LIN {X 0,Y 346.779,Z 652.941,A -85,B 0,C 180,E1 -23158.009,E2 -23158.009} C_VEL
LIN {X 0,Y 351.853,Z 640.47,A -85,B 0,C 180,E1 -23159.518,E2 -23159.518} C_VEL
LIN {X 0,Y 356.974,Z 626.516,A -85,B 0,C 180,E1 -23160.838,E2 -23160.838} C_VEL
LIN {X 0,Y 360.859,Z 614.191,A -85,B 0,C 180,E1 -23161.77,E2 -23161.77} C_VEL
LIN {X 0,Y 365.059,Z 598.938,A -85,B 0,C 180,E1 -23162.659,E2 -23162.659} C_VEL
LIN {X 0,Y 368.432,Z 583.567,A -85,B 0,C 180,E1 -23163.336,E2 -23163.336} C_VEL
LIN {X 0,Y 383.692,Z 497.433,A -85,B 0,C 180,E1 -23166.383,E2 -23166.383} C_VEL
LIN {X 0,Y 385.575,Z 481.18,A -85,B 0,C 180,E1 -23167.472,E2 -23167.472} C_VEL
LIN {X 0,Y 387.086,Z 465.883,A -85,B 0,C 180,E1 -23168.772,E2 -23168.772} C_VEL
LIN {X 0,Y 387.278,Z 463.542,A -85,B 0,C 180,E1 -23169.013,E2 -23169.013} C_VEL
LIN {X 0,Y 385.216,Z 461.451,A -85,B 0,C 180,E1 -23170.889,E2 -23170.889} C_VEL
LIN {X 0,Y 384.014,Z 460.701,A -85,B 0,C 180,E1 -23172.445,E2 -23172.445} C_VEL
LIN {X 0,Y 383.117,Z 460.948,A -85,B 0,C 180,E1 -23174.518,E2 -23174.518} C_VEL
LIN {X 0,Y 382.898,Z 462.38,A -85,B 0,C 180,E1 -23176.123,E2 -23176.123} C_VEL
LIN {X 0,Y 383.334,Z 465.723,A -85,B 0,C 180,E1 -23178.248,E2 -23178.248} C_VEL
LIN {X 0,Y 384.216,Z 470.909,A -85,B 0,C 180,E1 -23180.158,E2 -23180.158} C_VEL
LIN {X 0,Y 384.484,Z 473.066,A -85,B 0,C 180,E1 -23180.704,E2 -23180.704} C_VEL
LIN {X 0,Y 383.597,Z 487.714,A -85,B 0,C 180,E1 -23182.321,E2 -23182.321} C_VEL
LIN {X 0,Y 382.742,Z 502.862,A -85,B 0,C 180,E1 -23183.728,E2 -23183.728} C_VEL
LIN {X 0,Y 382.412,Z 505.3,A -85,B 0,C 180,E1 -23183.861,E2 -23183.861} C_VEL
LIN {X 0,Y 368.256,Z 585.492,A -85,B 0,C 180,E1 -23186.687,E2 -23186.687} C_VEL
LIN {X 0,Y 365.05,Z 599.465,A -85,B 0,C 180,E1 -23187.34,E2 -23187.34} C_VEL
LIN {X 0,Y 360.944,Z 614.223,A -85,B 0,C 180,E1 -23188.239,E2 -23188.239} C_VEL
LIN {X 0,Y 356.653,Z 627.599,A -85,B 0,C 180,E1 -23189.295,E2 -23189.295} C_VEL
LIN {X 0,Y 352.113,Z 639.917,A -85,B 0,C 180,E1 -23190.506,E2 -23190.506} C_VEL
LIN {X 0,Y 347.039,Z 652.252,A -85,B 0,C 180,E1 -23192.014,E2 -23192.014} C_VEL
LIN {X 0,Y 342.31,Z 662.634,A -85,B 0,C 180,E1 -23193.573,E2 -23193.573} C_VEL
LIN {X 0,Y 337.275,Z 672.679,A -85,B 0,C 180,E1 -23195.459,E2 -23195.459} C_VEL
LIN {X 0,Y 332.699,Z 681,A -85,B 0,C 180,E1 -23197.405,E2 -23197.405} C_VEL
LIN {X 0,Y 328.687,Z 687.815,A -85,B 0,C 180,E1 -23199.414,E2 -23199.414} C_VEL
LIN {X 0,Y 324.702,Z 693.917,A -85,B 0,C 180,E1 -23201.708,E2 -23201.708} C_VEL
LIN {X 0,Y 322.138,Z 697.676,A -85,B 0,C 180,E1 -23203.581,E2 -23203.581} C_VEL
LIN {X 0,Y 319.226,Z 701.269,A -85,B 0,C 180,E1 -23206.033,E2 -23206.033} C_VEL
LIN {X 0,Y 316.907,Z 703.492,A -85,B 0,C 180,E1 -23208.526,E2 -23208.526} C_VEL
LIN {X 0,Y 315.328,Z 704.371,A -85,B 0,C 180,E1 -23211.055,E2 -23211.055} C_VEL
LIN {X 0,Y 314.416,Z 703.91,A -85,B 0,C 180,E1 -23213.605,E2 -23213.605} C_VEL
LIN {X 0,Y 313.985,Z 702.1,A -85,B 0,C 180,E1 -23216.163,E2 -23216.163} C_VEL
LIN {X 0,Y 313.957,Z 698.885,A -85,B 0,C 180,E1 -23218.722,E2 -23218.722} C_VEL
LIN {X 0,Y 314.065,Z 695.439,A -85,B 0,C 180,E1 -23220.639,E2 -23220.639} C_VEL
LIN {X 0,Y 314.17,Z 691.067,A -85,B 0,C 180,E1 -23222.556,E2 -23222.556} C_VEL
LIN {X 0,Y 314.312,Z 684.61,A -85,B 0,C 180,E1 -23224.794,E2 -23224.794} C_VEL
LIN {X 0,Y 314.568,Z 676.533,A -85,B 0,C 180,E1 -23227.035,E2 -23227.035} C_VEL
LIN {X 0,Y 314.911,Z 668.051,A -85,B 0,C 180,E1 -23228.958,E2 -23228.958} C_VEL
LIN {X 0,Y 315.448,Z 657.845,A -85,B 0,C 180,E1 -23230.88,E2 -23230.88} C_VEL
LIN {X 0,Y 316.229,Z 646.555,A -85,B 0,C 180,E1 -23232.635,E2 -23232.635} C_VEL
LIN {X 0,Y 316.961,Z 634.117,A -85,B 0,C 180,E1 -23234.232,E2 -23234.232} C_VEL
LIN {X 0,Y 317.847,Z 620.529,A -85,B 0,C 180,E1 -23235.662,E2 -23235.662} C_VEL
LIN {X 0,Y 318.736,Z 606.233,A -85,B 0,C 180,E1 -23236.847,E2 -23236.847} C_VEL
LIN {X 0,Y 319.44,Z 591.469,A -85,B 0,C 180,E1 -23237.795,E2 -23237.795} C_VEL
LIN {X 0,Y 320.09,Z 576.464,A -85,B 0,C 180,E1 -23238.5,E2 -23238.5} C_VEL
LIN {X 0,Y 323.542,Z 476.916,A -85,B 0,C 180,E1 -23242.075,E2 -23242.075} C_VEL
LIN {X 0,Y 321.24,Z 448.747,A -85,B 0,C 180,E1 -23243.145,E2 -23243.145} C_VEL
LIN {X 0,Y 320.964,Z 439.558,A -85,B 0,C 180,E1 -23243.504,E2 -23243.504} C_VEL
LIN {X 0,Y 323.406,Z 412.958,A -85,B 0,C 180,E1 -23247.629,E2 -23247.629} C_VEL
LIN {X 0,Y 325.023,Z 396.535,A -85,B 0,C 180,E1 -23250.169,E2 -23250.169} C_VEL
LIN {X 0,Y 321.474,Z 379.818,A -85,B 0,C 180,E1 -23253.006,E2 -23253.006} C_VEL
LIN {X 0,Y 316.705,Z 358.595,A -85,B 0,C 180,E1 -23256.736,E2 -23256.736} C_VEL
LIN {X 0,Y 316.607,Z 358.599,A -85,B 0,C 180,E1 -23259.91,E2 -23259.91} C_VEL
LIN {X 0,Y 316.65,Z 358.6,A -85,B 0,C 180,E1 -23263.294,E2 -23263.294} C_VEL
LIN {X 0,Y 316.648,Z 358.598,A -85,B 0,C 180,E1 -23266.885,E2 -23266.885} C_VEL
LIN {X 0,Y 316.625,Z 358.599,A -85,B 0,C 180,E1 -23270.74,E2 -23270.74} C_VEL
LIN {X 0,Y 316.642,Z 358.594,A -85,B 0,C 180,E1 -23273.326,E2 -23273.326} C_VEL
LIN {X 0,Y 316.635,Z 358.596,A -85,B 0,C 180,E1 -23276.424,E2 -23276.424} C_VEL
LIN {X 0,Y 316.649,Z 358.592,A -85,B 0,C 180,E1 -23279.622,E2 -23279.622} C_VEL
LIN {X 0,Y 316.701,Z 358.593,A -85,B 0,C 180,E1 -23283.747,E2 -23283.747} C_VEL
LIN {X 0,Y 316.749,Z 358.588,A -85,B 0,C 180,E1 -23286.371,E2 -23286.371} C_VEL
LIN {X 0,Y 317.718,Z 361.443,A -85,B 0,C 180,E1 -23286.533,E2 -23286.533} C_VEL
LIN {X 0,Y 327.007,Z 380.664,A -85,B 0,C 180,E1 -23287.823,E2 -23287.823} C_VEL
LIN {X 0,Y 332.963,Z 394.934,A -85,B 0,C 180,E1 -23288.65,E2 -23288.65} C_VEL
LIN {X 0,Y 331.321,Z 465.528,A -85,B 0,C 180,E1 -23290.164,E2 -23290.164} C_VEL
LIN {X 0,Y 331.032,Z 481.627,A -85,B 0,C 180,E1 -23290.614,E2 -23290.614} C_VEL
LIN {X 0,Y 330.468,Z 495.129,A -85,B 0,C 180,E1 -23291.222,E2 -23291.222} C_VEL
LIN {X 0,Y 329.533,Z 508.415,A -85,B 0,C 180,E1 -23292.049,E2 -23292.049} C_VEL
LIN {X 0,Y 328.22,Z 521.311,A -85,B 0,C 180,E1 -23293.096,E2 -23293.096} C_VEL
LIN {X 0,Y 326.791,Z 534.282,A -85,B 0,C 180,E1 -23294.459,E2 -23294.459} C_VEL
LIN {X 0,Y 325.343,Z 544.759,A -85,B 0,C 180,E1 -23295.804,E2 -23295.804} C_VEL
LIN {X 0,Y 323.521,Z 555.634,A -85,B 0,C 180,E1 -23297.496,E2 -23297.496} C_VEL
LIN {X 0,Y 321.797,Z 565.3,A -85,B 0,C 180,E1 -23299.338,E2 -23299.338} C_VEL
LIN {X 0,Y 320.333,Z 573.323,A -85,B 0,C 180,E1 -23301.196,E2 -23301.196} C_VEL
LIN {X 0,Y 319.085,Z 580.021,A -85,B 0,C 180,E1 -23303.066,E2 -23303.066} C_VEL
LIN {X 0,Y 318.016,Z 585.608,A -85,B 0,C 180,E1 -23304.946,E2 -23304.946} C_VEL
LIN {X 0,Y 317.008,Z 591.463,A -85,B 0,C 180,E1 -23307.467,E2 -23307.467} C_VEL
LIN {X 0,Y 316.393,Z 595.771,A -85,B 0,C 180,E1 -23310,E2 -23310} C_VEL
LIN {X 0,Y 315.984,Z 598.694,A -85,B 0,C 180,E1 -23312.541,E2 -23312.541} C_VEL
LIN {X 0,Y 316.031,Z 600.28,A -85,B 0,C 180,E1 -23315.086,E2 -23315.086} C_VEL
LIN {X 0,Y 316.305,Z 600.584,A -85,B 0,C 180,E1 -23317.636,E2 -23317.636} C_VEL
LIN {X 0,Y 316.886,Z 599.6,A -85,B 0,C 180,E1 -23320.186,E2 -23320.186} C_VEL
LIN {X 0,Y 317.872,Z 597.292,A -85,B 0,C 180,E1 -23322.73,E2 -23322.73} C_VEL
LIN {X 0,Y 319.35,Z 593.581,A -85,B 0,C 180,E1 -23325.26,E2 -23325.26} C_VEL
LIN {X 0,Y 321.139,Z 588.317,A -85,B 0,C 180,E1 -23327.78,E2 -23327.78} C_VEL
LIN {X 0,Y 322.768,Z 583.279,A -85,B 0,C 180,E1 -23329.656,E2 -23329.656} C_VEL
LIN {X 0,Y 325.037,Z 575.645,A -85,B 0,C 180,E1 -23331.923,E2 -23331.923} C_VEL
LIN {X 0,Y 327.491,Z 566.918,A -85,B 0,C 180,E1 -23333.978,E2 -23333.978} C_VEL
LIN {X 0,Y 329.941,Z 557.378,A -85,B 0,C 180,E1 -23335.799,E2 -23335.799} C_VEL
LIN {X 0,Y 332.282,Z 546.761,A -85,B 0,C 180,E1 -23337.46,E2 -23337.46} C_VEL
LIN {X 0,Y 334.603,Z 534.957,A -85,B 0,C 180,E1 -23338.953,E2 -23338.953} C_VEL
LIN {X 0,Y 336.61,Z 523.311,A -85,B 0,C 180,E1 -23340.134,E2 -23340.134} C_VEL
LIN {X 0,Y 338.141,Z 510.547,A -85,B 0,C 180,E1 -23341.189,E2 -23341.189} C_VEL
LIN {X 0,Y 339.438,Z 497.149,A -85,B 0,C 180,E1 -23342.03,E2 -23342.03} C_VEL
LIN {X 0,Y 340.324,Z 482.787,A -85,B 0,C 180,E1 -23342.674,E2 -23342.674} C_VEL
LIN {X 0,Y 340.732,Z 467.217,A -85,B 0,C 180,E1 -23343.114,E2 -23343.114} C_VEL
LIN {X 0,Y 342.688,Z 407.141,A -85,B 0,C 180,E1 -23344.365,E2 -23344.365} C_VEL
LIN {X 0,Y 334.807,Z 391.079,A -85,B 0,C 180,E1 -23345.625,E2 -23345.625} C_VEL
LIN {X 0,Y 324.967,Z 373.249,A -85,B 0,C 180,E1 -23347.256,E2 -23347.256} C_VEL
LIN {X 0,Y 318.296,Z 362.362,A -85,B 0,C 180,E1 -23348.406,E2 -23348.406} C_VEL
LIN {X 0,Y 316.879,Z 359.863,A -85,B 0,C 180,E1 -23348.664,E2 -23348.664} C_VEL
LIN {X 0,Y 316.605,Z 358.608,A -85,B 0,C 180,E1 -23348.766,E2 -23348.766} C_VEL
LIN {X 0,Y 316.591,Z 358.608,A -85,B 0,C 180,E1 -23351.586,E2 -23351.586} C_VEL
LIN {X 0,Y 316.61,Z 358.6,A -85,B 0,C 180,E1 -23355.068,E2 -23355.068} C_VEL
LIN {X 0,Y 316.606,Z 358.602,A -85,B 0,C 180,E1 -23358.782,E2 -23358.782} C_VEL
LIN {X 0,Y 316.63,Z 358.554,A -85,B 0,C 180,E1 -23362.787,E2 -23362.787} C_VEL
LIN {X 0,Y 316.621,Z 358.596,A -85,B 0,C 180,E1 -23366.422,E2 -23366.422} C_VEL
LIN {X 0,Y 316.626,Z 358.587,A -85,B 0,C 180,E1 -23369.629,E2 -23369.629} C_VEL
LIN {X 0,Y 316.684,Z 358.581,A -85,B 0,C 180,E1 -23373.745,E2 -23373.745} C_VEL
LIN {X 0,Y 316.719,Z 358.59,A -85,B 0,C 180,E1 -23376.824,E2 -23376.824} C_VEL
LIN {X 0,Y 322.641,Z 381.681,A -85,B 0,C 180,E1 -23377.798,E2 -23377.798} C_VEL
LIN {X 0,Y 322.664,Z 387.019,A -85,B 0,C 180,E1 -23377.988,E2 -23377.988} C_VEL
LIN {X 0,Y 321.766,Z 392.772,A -85,B 0,C 180,E1 -23378.173,E2 -23378.173} C_VEL
LIN {X 0,Y 315.268,Z 411.293,A -85,B 0,C 180,E1 -23378.723,E2 -23378.723} C_VEL
LIN {X 0,Y 314.476,Z 417.043,A -85,B 0,C 180,E1 -23378.922,E2 -23378.922} C_VEL
LIN {X 0,Y 313.091,Z 476.776,A -85,B 0,C 180,E1 -23381.113,E2 -23381.113} C_VEL
LIN {X 0,Y 312.579,Z 491.416,A -85,B 0,C 180,E1 -23381.885,E2 -23381.885} C_VEL
LIN {X 0,Y 312.014,Z 505.448,A -85,B 0,C 180,E1 -23382.863,E2 -23382.863} C_VEL
LIN {X 0,Y 311.237,Z 520.037,A -85,B 0,C 180,E1 -23384.164,E2 -23384.164} C_VEL
LIN {X 0,Y 310.556,Z 533.361,A -85,B 0,C 180,E1 -23385.635,E2 -23385.635} C_VEL
LIN {X 0,Y 309.939,Z 545.605,A -85,B 0,C 180,E1 -23387.27,E2 -23387.27} C_VEL
LIN {X 0,Y 309.213,Z 557.66,A -85,B 0,C 180,E1 -23389.229,E2 -23389.229} C_VEL
LIN {X 0,Y 308.697,Z 567.679,A -85,B 0,C 180,E1 -23391.19,E2 -23391.19} C_VEL
LIN {X 0,Y 308.33,Z 577.376,A -85,B 0,C 180,E1 -23393.478,E2 -23393.478} C_VEL
LIN {X 0,Y 308.286,Z 585.271,A -85,B 0,C 180,E1 -23395.765,E2 -23395.765} C_VEL
LIN {X 0,Y 308.365,Z 591.806,A -85,B 0,C 180,E1 -23398.112,E2 -23398.112} C_VEL
LIN {X 0,Y 308.83,Z 597.364,A -85,B 0,C 180,E1 -23400.649,E2 -23400.649} C_VEL
LIN {X 0,Y 309.447,Z 600.59,A -85,B 0,C 180,E1 -23402.594,E2 -23402.594} C_VEL
LIN {X 0,Y 310.787,Z 603.654,A -85,B 0,C 180,E1 -23405.172,E2 -23405.172} C_VEL
LIN {X 0,Y 312.509,Z 605.336,A -85,B 0,C 180,E1 -23407.728,E2 -23407.728} C_VEL
LIN {X 0,Y 314.673,Z 605.643,A -85,B 0,C 180,E1 -23410.257,E2 -23410.257} C_VEL
LIN {X 0,Y 317.708,Z 604.49,A -85,B 0,C 180,E1 -23412.736,E2 -23412.736} C_VEL
LIN {X 0,Y 321.376,Z 601.907,A -85,B 0,C 180,E1 -23415.161,E2 -23415.161} C_VEL
LIN {X 0,Y 325.315,Z 597.923,A -85,B 0,C 180,E1 -23417.544,E2 -23417.544} C_VEL
LIN {X 0,Y 328.569,Z 593.917,A -85,B 0,C 180,E1 -23419.295,E2 -23419.295} C_VEL
LIN {X 0,Y 333.406,Z 587.105,A -85,B 0,C 180,E1 -23421.571,E2 -23421.571} C_VEL
LIN {X 0,Y 337.979,Z 579.557,A -85,B 0,C 180,E1 -23423.512,E2 -23423.512} C_VEL
LIN {X 0,Y 342.881,Z 570.267,A -85,B 0,C 180,E1 -23425.403,E2 -23425.403} C_VEL
LIN {X 0,Y 347.411,Z 560.641,A -85,B 0,C 180,E1 -23426.977,E2 -23426.977} C_VEL
LIN {X 0,Y 352.14,Z 549.032,A -85,B 0,C 180,E1 -23428.515,E2 -23428.515} C_VEL
LIN {X 0,Y 356.656,Z 536.172,A -85,B 0,C 180,E1 -23429.89,E2 -23429.89} C_VEL
LIN {X 0,Y 360.336,Z 523.4,A -85,B 0,C 180,E1 -23431.006,E2 -23431.006} C_VEL
LIN {X 0,Y 363.682,Z 509.402,A -85,B 0,C 180,E1 -23431.981,E2 -23431.981} C_VEL
LIN {X 0,Y 366.369,Z 495.047,A -85,B 0,C 180,E1 -23432.767,E2 -23432.767} C_VEL
LIN {X 0,Y 370.41,Z 469.275,A -85,B 0,C 180,E1 -23433.806,E2 -23433.806} C_VEL
LIN {X 0,Y 375.351,Z 441.241,A -85,B 0,C 180,E1 -23434.806,E2 -23434.806} C_VEL
LIN {X 0,Y 373.14,Z 436.29,A -85,B 0,C 180,E1 -23436.453,E2 -23436.453} C_VEL
LIN {X 0,Y 371.66,Z 433.21,A -85,B 0,C 180,E1 -23437.804,E2 -23437.804} C_VEL
LIN {X 0,Y 370.173,Z 429.982,A -85,B 0,C 180,E1 -23439.676,E2 -23439.676} C_VEL
LIN {X 0,Y 368.834,Z 428.602,A -85,B 0,C 180,E1 -23442.214,E2 -23442.214} C_VEL
LIN {X 0,Y 368.77,Z 428.453,A -85,B 0,C 180,E1 -23444.198,E2 -23444.198} C_VEL
LIN {X 0,Y 369.948,Z 429.972,A -85,B 0,C 180,E1 -23447.03,E2 -23447.03} C_VEL
LIN {X 0,Y 371.094,Z 432.974,A -85,B 0,C 180,E1 -23448.705,E2 -23448.705} C_VEL
LIN {X 0,Y 371.308,Z 443.447,A -85,B 0,C 180,E1 -23450.524,E2 -23450.524} C_VEL
LIN {X 0,Y 370.005,Z 459.779,A -85,B 0,C 180,E1 -23451.954,E2 -23451.954} C_VEL
LIN {X 0,Y 368.744,Z 476.184,A -85,B 0,C 180,E1 -23453.226,E2 -23453.226} C_VEL
LIN {X 0,Y 367.73,Z 487.498,A -85,B 0,C 180,E1 -23453.981,E2 -23453.981} C_VEL
LIN {X 0,Y 366.638,Z 496.863,A -85,B 0,C 180,E1 -23454.488,E2 -23454.488} C_VEL
LIN {X 0,Y 360.902,Z 530.902,A -85,B 0,C 180,E1 -23455.705,E2 -23455.705} C_VEL
LIN {X 0,Y 356.785,Z 548.297,A -85,B 0,C 180,E1 -23456.485,E2 -23456.485} C_VEL
LIN {X 0,Y 352.248,Z 563.594,A -85,B 0,C 180,E1 -23457.358,E2 -23457.358} C_VEL
LIN {X 0,Y 347.42,Z 577.531,A -85,B 0,C 180,E1 -23458.386,E2 -23458.386} C_VEL
LIN {X 0,Y 341.838,Z 591.573,A -85,B 0,C 180,E1 -23459.696,E2 -23459.696} C_VEL
LIN {X 0,Y 336.493,Z 603.77,A -85,B 0,C 180,E1 -23461.124,E2 -23461.124} C_VEL
LIN {X 0,Y 331.55,Z 614.197,A -85,B 0,C 180,E1 -23462.645,E2 -23462.645} C_VEL
LIN {X 0,Y 326.244,Z 624.904,A -85,B 0,C 180,E1 -23464.57,E2 -23464.57} C_VEL
LIN {X 0,Y 321.587,Z 633.763,A -85,B 0,C 180,E1 -23466.578,E2 -23466.578} C_VEL
LIN {X 0,Y 317.657,Z 641.179,A -85,B 0,C 180,E1 -23468.664,E2 -23468.664} C_VEL
LIN {X 0,Y 314.652,Z 646.488,A -85,B 0,C 180,E1 -23470.493,E2 -23470.493} C_VEL
LIN {X 0,Y 311.633,Z 652.249,A -85,B 0,C 180,E1 -23473.01,E2 -23473.01} C_VEL
LIN {X 0,Y 309.58,Z 656.596,A -85,B 0,C 180,E1 -23475.588,E2 -23475.588} C_VEL
LIN {X 0,Y 308.34,Z 659.625,A -85,B 0,C 180,E1 -23478.202,E2 -23478.202} C_VEL
LIN {X 0,Y 308.143,Z 660.826,A -85,B 0,C 180,E1 -23479.729,E2 -23479.729} C_VEL
LIN {X 0,Y 307.758,Z 669.853,A -85,B 0,C 180,E1 -23481.492,E2 -23481.492} C_VEL
LIN {X 0,Y 307.479,Z 678.288,A -85,B 0,C 180,E1 -23483.46,E2 -23483.46} C_VEL
LIN {X 0,Y 307.33,Z 686.328,A -85,B 0,C 180,E1 -23485.752,E2 -23485.752} C_VEL
LIN {X 0,Y 307.193,Z 692.677,A -85,B 0,C 180,E1 -23488.04,E2 -23488.04} C_VEL
LIN {X 0,Y 307.15,Z 696.963,A -85,B 0,C 180,E1 -23490,E2 -23490} C_VEL
LIN {X 0,Y 306.964,Z 701.209,A -85,B 0,C 180,E1 -23492.616,E2 -23492.616} C_VEL
LIN {X 0,Y 307.071,Z 703.981,A -85,B 0,C 180,E1 -23495.235,E2 -23495.235} C_VEL
LIN {X 0,Y 307.682,Z 705.368,A -85,B 0,C 180,E1 -23497.85,E2 -23497.85} C_VEL
LIN {X 0,Y 308.888,Z 705.414,A -85,B 0,C 180,E1 -23500.452,E2 -23500.452} C_VEL
LIN {X 0,Y 310.84,Z 704.125,A -85,B 0,C 180,E1 -23503.023,E2 -23503.023} C_VEL
LIN {X 0,Y 313.636,Z 701.476,A -85,B 0,C 180,E1 -23505.545,E2 -23505.545} C_VEL
LIN {X 0,Y 316.707,Z 697.478,A -85,B 0,C 180,E1 -23508.037,E2 -23508.037} C_VEL
LIN {X 0,Y 320.721,Z 691.969,A -85,B 0,C 180,E1 -23510.453,E2 -23510.453} C_VEL
LIN {X 0,Y 325.464,Z 684.838,A -85,B 0,C 180,E1 -23512.792,E2 -23512.792} C_VEL
LIN {X 0,Y 330.082,Z 677.116,A -85,B 0,C 180,E1 -23514.778,E2 -23514.778} C_VEL
LIN {X 0,Y 335.287,Z 667.758,A -85,B 0,C 180,E1 -23516.689,E2 -23516.689} C_VEL
LIN {X 0,Y 340.088,Z 658.186,A -85,B 0,C 180,E1 -23518.275,E2 -23518.275} C_VEL
LIN {X 0,Y 345.725,Z 645.746,A -85,B 0,C 180,E1 -23519.928,E2 -23519.928} C_VEL
LIN {X 0,Y 350.346,Z 634.318,A -85,B 0,C 180,E1 -23521.152,E2 -23521.152} C_VEL
LIN {X 0,Y 355.301,Z 620.631,A -85,B 0,C 180,E1 -23522.327,E2 -23522.327} C_VEL
LIN {X 0,Y 360.184,Z 604.828,A -85,B 0,C 180,E1 -23523.357,E2 -23523.357} C_VEL
LIN {X 0,Y 363.719,Z 591.16,A -85,B 0,C 180,E1 -23524.034,E2 -23524.034} C_VEL
LIN {X 0,Y 367.59,Z 571.441,A -85,B 0,C 180,E1 -23524.782,E2 -23524.782} C_VEL
LIN {X 0,Y 381.113,Z 498.793,A -85,B 0,C 180,E1 -23527.362,E2 -23527.362} C_VEL
LIN {X 0,Y 383.099,Z 483.725,A -85,B 0,C 180,E1 -23528.391,E2 -23528.391} C_VEL
LIN {X 0,Y 384.77,Z 469.789,A -85,B 0,C 180,E1 -23529.579,E2 -23529.579} C_VEL
LIN {X 0,Y 383.357,Z 468.269,A -85,B 0,C 180,E1 -23530.972,E2 -23530.972} C_VEL
LIN {X 0,Y 382.078,Z 467.548,A -85,B 0,C 180,E1 -23532.711,E2 -23532.711} C_VEL
LIN {X 0,Y 381.318,Z 467.919,A -85,B 0,C 180,E1 -23534.616,E2 -23534.616} C_VEL
LIN {X 0,Y 381.122,Z 469.709,A -85,B 0,C 180,E1 -23536.392,E2 -23536.392} C_VEL
LIN {X 0,Y 381.417,Z 472.559,A -85,B 0,C 180,E1 -23538.079,E2 -23538.079} C_VEL
LIN {X 0,Y 382.066,Z 477.105,A -85,B 0,C 180,E1 -23539.76,E2 -23539.76} C_VEL
LIN {X 0,Y 382.12,Z 478.457,A -85,B 0,C 180,E1 -23540.064,E2 -23540.064} C_VEL
LIN {X 0,Y 380.815,Z 494.198,A -85,B 0,C 180,E1 -23541.784,E2 -23541.784} C_VEL
LIN {X 0,Y 379.927,Z 505.742,A -85,B 0,C 180,E1 -23542.854,E2 -23542.854} C_VEL
LIN {X 0,Y 367.019,Z 575.904,A -85,B 0,C 180,E1 -23545.322,E2 -23545.322} C_VEL
LIN {X 0,Y 363.346,Z 593.162,A -85,B 0,C 180,E1 -23546.01,E2 -23546.01} C_VEL
LIN {X 0,Y 359.038,Z 609.143,A -85,B 0,C 180,E1 -23546.89,E2 -23546.89} C_VEL
LIN {X 0,Y 354.944,Z 621.931,A -85,B 0,C 180,E1 -23547.804,E2 -23547.804} C_VEL
LIN {X 0,Y 350.056,Z 635.127,A -85,B 0,C 180,E1 -23548.986,E2 -23548.986} C_VEL
LIN {X 0,Y 345.053,Z 647.242,A -85,B 0,C 180,E1 -23550.343,E2 -23550.343} C_VEL
LIN {X 0,Y 340.342,Z 657.483,A -85,B 0,C 180,E1 -23551.748,E2 -23551.748} C_VEL
LIN {X 0,Y 334.758,Z 668.398,A -85,B 0,C 180,E1 -23553.6,E2 -23553.6} C_VEL
LIN {X 0,Y 329.702,Z 677.411,A -85,B 0,C 180,E1 -23555.527,E2 -23555.527} C_VEL
LIN {X 0,Y 325.727,Z 683.918,A -85,B 0,C 180,E1 -23557.228,E2 -23557.228} C_VEL
LIN {X 0,Y 321.099,Z 690.959,A -85,B 0,C 180,E1 -23559.573,E2 -23559.573} C_VEL
LIN {X 0,Y 316.996,Z 696.44,A -85,B 0,C 180,E1 -23561.98,E2 -23561.98} C_VEL
LIN {X 0,Y 313.898,Z 700.4,A -85,B 0,C 180,E1 -23564.469,E2 -23564.469} C_VEL
LIN {X 0,Y 311.068,Z 703.028,A -85,B 0,C 180,E1 -23566.987,E2 -23566.987} C_VEL
LIN {X 0,Y 309.051,Z 704.298,A -85,B 0,C 180,E1 -23569.554,E2 -23569.554} C_VEL
LIN {X 0,Y 307.759,Z 704.237,A -85,B 0,C 180,E1 -23572.152,E2 -23572.152} C_VEL
LIN {X 0,Y 307.078,Z 702.839,A -85,B 0,C 180,E1 -23574.765,E2 -23574.765} C_VEL
LIN {X 0,Y 306.869,Z 700.065,A -85,B 0,C 180,E1 -23577.384,E2 -23577.384} C_VEL
LIN {X 0,Y 306.986,Z 695.832,A -85,B 0,C 180,E1 -23580,E2 -23580} C_VEL
LIN {X 0,Y 307.097,Z 691.59,A -85,B 0,C 180,E1 -23581.961,E2 -23581.961} C_VEL
LIN {X 0,Y 307.279,Z 685.311,A -85,B 0,C 180,E1 -23584.249,E2 -23584.249} C_VEL
LIN {X 0,Y 307.46,Z 677.251,A -85,B 0,C 180,E1 -23586.576,E2 -23586.576} C_VEL
LIN {X 0,Y 307.848,Z 667.58,A -85,B 0,C 180,E1 -23588.835,E2 -23588.835} C_VEL
LIN {X 0,Y 308.407,Z 657.294,A -85,B 0,C 180,E1 -23590.8,E2 -23590.8} C_VEL
LIN {X 0,Y 309.188,Z 645.655,A -85,B 0,C 180,E1 -23592.635,E2 -23592.635} C_VEL
LIN {X 0,Y 309.896,Z 633.374,A -85,B 0,C 180,E1 -23594.23,E2 -23594.23} C_VEL
LIN {X 0,Y 310.831,Z 619.593,A -85,B 0,C 180,E1 -23595.689,E2 -23595.689} C_VEL
LIN {X 0,Y 311.678,Z 605.115,A -85,B 0,C 180,E1 -23596.903,E2 -23596.903} C_VEL
LIN {X 0,Y 312.371,Z 590.156,A -85,B 0,C 180,E1 -23597.874,E2 -23597.874} C_VEL
LIN {X 0,Y 313.093,Z 573.682,A -85,B 0,C 180,E1 -23598.633,E2 -23598.633} C_VEL
LIN {X 0,Y 316.466,Z 477.377,A -85,B 0,C 180,E1 -23602.199,E2 -23602.199} C_VEL
LIN {X 0,Y 314.199,Z 448.926,A -85,B 0,C 180,E1 -23603.31,E2 -23603.31} C_VEL
LIN {X 0,Y 313.934,Z 439.598,A -85,B 0,C 180,E1 -23603.68,E2 -23603.68} C_VEL
LIN {X 0,Y 316.358,Z 414.017,A -85,B 0,C 180,E1 -23607.708,E2 -23607.708} C_VEL
LIN {X 0,Y 317.988,Z 397.796,A -85,B 0,C 180,E1 -23610.257,E2 -23610.257} C_VEL
LIN {X 0,Y 315.094,Z 383.863,A -85,B 0,C 180,E1 -23612.654,E2 -23612.654} C_VEL
LIN {X 0,Y 310.71,Z 364.228,A -85,B 0,C 180,E1 -23616.117,E2 -23616.117} C_VEL
LIN {X 0,Y 309.662,Z 359.473,A -85,B 0,C 180,E1 -23616.997,E2 -23616.997} C_VEL
LIN {X 0,Y 309.591,Z 359.473,A -85,B 0,C 180,E1 -23621.005,E2 -23621.005} C_VEL
LIN {X 0,Y 309.61,Z 359.476,A -85,B 0,C 180,E1 -23624.534,E2 -23624.534} C_VEL
LIN {X 0,Y 309.593,Z 359.478,A -85,B 0,C 180,E1 -23628.299,E2 -23628.299} C_VEL
LIN {X 0,Y 309.609,Z 359.477,A -85,B 0,C 180,E1 -23632.357,E2 -23632.357} C_VEL
LIN {X 0,Y 309.593,Z 359.476,A -85,B 0,C 180,E1 -23635.555,E2 -23635.555} C_VEL
LIN {X 0,Y 309.606,Z 359.464,A -85,B 0,C 180,E1 -23639.284,E2 -23639.284} C_VEL
LIN {X 0,Y 309.641,Z 359.473,A -85,B 0,C 180,E1 -23643.101,E2 -23643.101} C_VEL
LIN {X 0,Y 309.669,Z 359.469,A -85,B 0,C 180,E1 -23645.699,E2 -23645.699} C_VEL
LIN {X 0,Y 310.783,Z 362.472,A -85,B 0,C 180,E1 -23645.904,E2 -23645.904} C_VEL
LIN {X 0,Y 320.548,Z 382.539,A -85,B 0,C 180,E1 -23647.309,E2 -23647.309} C_VEL
LIN {X 0,Y 326.56,Z 396.904,A -85,B 0,C 180,E1 -23648.173,E2 -23648.173} C_VEL
LIN {X 0,Y 324.818,Z 464.966,A -85,B 0,C 180,E1 -23649.652,E2 -23649.652} C_VEL
LIN {X 0,Y 324.54,Z 480.842,A -85,B 0,C 180,E1 -23650.087,E2 -23650.087} C_VEL
LIN {X 0,Y 323.967,Z 494.854,A -85,B 0,C 180,E1 -23650.707,E2 -23650.707} C_VEL
LIN {X 0,Y 322.977,Z 508.959,A -85,B 0,C 180,E1 -23651.59,E2 -23651.59} C_VEL
LIN {X 0,Y 321.687,Z 521.072,A -85,B 0,C 180,E1 -23652.579,E2 -23652.579} C_VEL
LIN {X 0,Y 320.379,Z 532.973,A -85,B 0,C 180,E1 -23653.814,E2 -23653.814} C_VEL
LIN {X 0,Y 318.861,Z 543.972,A -85,B 0,C 180,E1 -23655.21,E2 -23655.21} C_VEL
LIN {X 0,Y 316.995,Z 554.996,A -85,B 0,C 180,E1 -23656.91,E2 -23656.91} C_VEL
LIN {X 0,Y 315.153,Z 564.901,A -85,B 0,C 180,E1 -23658.786,E2 -23658.786} C_VEL
LIN {X 0,Y 313.611,Z 573.123,A -85,B 0,C 180,E1 -23660.681,E2 -23660.681} C_VEL
LIN {X 0,Y 312.091,Z 580.985,A -85,B 0,C 180,E1 -23662.91,E2 -23662.91} C_VEL
LIN {X 0,Y 311.005,Z 586.539,A -85,B 0,C 180,E1 -23664.832,E2 -23664.832} C_VEL
LIN {X 0,Y 309.978,Z 592.35,A -85,B 0,C 180,E1 -23667.41,E2 -23667.41} C_VEL
LIN {X 0,Y 309.325,Z 596.627,A -85,B 0,C 180,E1 -23670,E2 -23670} C_VEL
LIN {X 0,Y 308.935,Z 599.516,A -85,B 0,C 180,E1 -23672.599,E2 -23672.599} C_VEL
LIN {X 0,Y 308.995,Z 601.071,A -85,B 0,C 180,E1 -23675.203,E2 -23675.203} C_VEL
LIN {X 0,Y 309.288,Z 601.346,A -85,B 0,C 180,E1 -23677.81,E2 -23677.81} C_VEL
LIN {X 0,Y 309.908,Z 600.331,A -85,B 0,C 180,E1 -23680.417,E2 -23680.417} C_VEL
LIN {X 0,Y 310.971,Z 597.989,A -85,B 0,C 180,E1 -23683.017,E2 -23683.017} C_VEL
LIN {X 0,Y 312.483,Z 594.241,A -85,B 0,C 180,E1 -23685.604,E2 -23685.604} C_VEL
LIN {X 0,Y 314.358,Z 588.93,A -85,B 0,C 180,E1 -23688.177,E2 -23688.177} C_VEL
LIN {X 0,Y 316.061,Z 583.869,A -85,B 0,C 180,E1 -23690.091,E2 -23690.091} C_VEL
LIN {X 0,Y 318.33,Z 576.573,A -85,B 0,C 180,E1 -23692.298,E2 -23692.298} C_VEL
LIN {X 0,Y 320.604,Z 568.858,A -85,B 0,C 180,E1 -23694.183,E2 -23694.183} C_VEL
LIN {X 0,Y 323.088,Z 559.56,A -85,B 0,C 180,E1 -23696.041,E2 -23696.041} C_VEL
LIN {X 0,Y 325.558,Z 549.225,A -85,B 0,C 180,E1 -23697.728,E2 -23697.728} C_VEL
LIN {X 0,Y 327.647,Z 539.067,A -85,B 0,C 180,E1 -23699.101,E2 -23699.101} C_VEL
LIN {X 0,Y 329.966,Z 526.602,A -85,B 0,C 180,E1 -23700.452,E2 -23700.452} C_VEL
LIN {X 0,Y 331.604,Z 514.494,A -85,B 0,C 180,E1 -23701.52,E2 -23701.52} C_VEL
LIN {X 0,Y 333.051,Z 500.538,A -85,B 0,C 180,E1 -23702.47,E2 -23702.47} C_VEL
LIN {X 0,Y 334.067,Z 486.744,A -85,B 0,C 180,E1 -23703.148,E2 -23703.148} C_VEL
LIN {X 0,Y 334.552,Z 472.312,A -85,B 0,C 180,E1 -23703.623,E2 -23703.623} C_VEL
LIN {X 0,Y 336.632,Z 409.302,A -85,B 0,C 180,E1 -23704.965,E2 -23704.965} C_VEL
LIN {X 0,Y 329.186,Z 394.16,A -85,B 0,C 180,E1 -23706.198,E2 -23706.198} C_VEL
LIN {X 0,Y 319.879,Z 377.285,A -85,B 0,C 180,E1 -23707.792,E2 -23707.792} C_VEL
LIN {X 0,Y 311.554,Z 363.621,A -85,B 0,C 180,E1 -23709.288,E2 -23709.288} C_VEL
LIN {X 0,Y 309.943,Z 361.107,A -85,B 0,C 180,E1 -23709.587,E2 -23709.587} C_VEL
LIN {X 0,Y 309.523,Z 359.486,A -85,B 0,C 180,E1 -23709.698,E2 -23709.698} C_VEL
LIN {X 0,Y 309.577,Z 359.486,A -85,B 0,C 180,E1 -23713.611,E2 -23713.611} C_VEL
LIN {X 0,Y 309.573,Z 359.478,A -85,B 0,C 180,E1 -23717.251,E2 -23717.251} C_VEL
LIN {X 0,Y 309.529,Z 359.475,A -85,B 0,C 180,E1 -23720.681,E2 -23720.681} C_VEL
LIN {X 0,Y 309.573,Z 359.433,A -85,B 0,C 180,E1 -23723.964,E2 -23723.964} C_VEL
LIN {X 0,Y 309.614,Z 359.472,A -85,B 0,C 180,E1 -23727.114,E2 -23727.114} C_VEL
LIN {X 0,Y 309.559,Z 359.47,A -85,B 0,C 180,E1 -23730.145,E2 -23730.145} C_VEL
LIN {X 0,Y 309.622,Z 359.465,A -85,B 0,C 180,E1 -23733.098,E2 -23733.098} C_VEL
LIN {X 0,Y 309.684,Z 359.491,A -85,B 0,C 180,E1 -23736.703,E2 -23736.703} C_VEL
LIN {X 0,Y 315.272,Z 381.677,A -85,B 0,C 180,E1 -23737.644,E2 -23737.644} C_VEL
LIN {X 0,Y 315.703,Z 384.262,A -85,B 0,C 180,E1 -23737.747,E2 -23737.747} C_VEL
LIN {X 0,Y 314.476,Z 417.043,A -85,B 0,C 180,E1 -23738.922,E2 -23738.922} C_VEL
LIN {X 0,Y 313.661,Z 422.799,A -85,B 0,C 180,E1 -23739.12,E2 -23739.12} C_VEL
LIN {X 0,Y 307.271,Z 441.334,A -85,B 0,C 180,E1 -23739.724,E2 -23739.724} C_VEL
LIN {X 0,Y 306.552,Z 447.09,A -85,B 0,C 180,E1 -23739.933,E2 -23739.933} C_VEL
LIN {X 0,Y 305.983,Z 478.878,A -85,B 0,C 180,E1 -23741.178,E2 -23741.178} C_VEL
LIN {X 0,Y 305.383,Z 494.404,A -85,B 0,C 180,E1 -23742.048,E2 -23742.048} C_VEL
LIN {X 0,Y 304.748,Z 508.843,A -85,B 0,C 180,E1 -23743.131,E2 -23743.131} C_VEL
LIN {X 0,Y 303.984,Z 522.956,A -85,B 0,C 180,E1 -23744.462,E2 -23744.462} C_VEL
LIN {X 0,Y 303.311,Z 535.934,A -85,B 0,C 180,E1 -23745.971,E2 -23745.971} C_VEL
LIN {X 0,Y 302.615,Z 548.818,A -85,B 0,C 180,E1 -23747.806,E2 -23747.806} C_VEL
LIN {X 0,Y 301.996,Z 559.59,A -85,B 0,C 180,E1 -23749.644,E2 -23749.644} C_VEL
LIN {X 0,Y 301.502,Z 569.477,A -85,B 0,C 180,E1 -23751.651,E2 -23751.651} C_VEL
LIN {X 0,Y 301.195,Z 578.958,A -85,B 0,C 180,E1 -23753.993,E2 -23753.993} C_VEL
LIN {X 0,Y 301.198,Z 586.728,A -85,B 0,C 180,E1 -23756.333,E2 -23756.333} C_VEL
LIN {X 0,Y 301.363,Z 593.024,A -85,B 0,C 180,E1 -23758.668,E2 -23758.668} C_VEL
LIN {X 0,Y 301.95,Z 598.65,A -85,B 0,C 180,E1 -23761.329,E2 -23761.329} C_VEL
LIN {X 0,Y 302.979,Z 602.705,A -85,B 0,C 180,E1 -23763.977,E2 -23763.977} C_VEL
LIN {X 0,Y 304.607,Z 605.33,A -85,B 0,C 180,E1 -23766.602,E2 -23766.602} C_VEL
LIN {X 0,Y 306.596,Z 606.606,A -85,B 0,C 180,E1 -23769.202,E2 -23769.202} C_VEL
LIN {X 0,Y 309.248,Z 606.507,A -85,B 0,C 180,E1 -23771.762,E2 -23771.762} C_VEL
LIN {X 0,Y 312.824,Z 604.97,A -85,B 0,C 180,E1 -23774.258,E2 -23774.258} C_VEL
LIN {X 0,Y 316.745,Z 602.045,A -85,B 0,C 180,E1 -23776.707,E2 -23776.707} C_VEL
LIN {X 0,Y 321.055,Z 597.649,A -85,B 0,C 180,E1 -23779.102,E2 -23779.102} C_VEL
LIN {X 0,Y 325.964,Z 591.664,A -85,B 0,C 180,E1 -23781.426,E2 -23781.426} C_VEL
LIN {X 0,Y 330.593,Z 584.967,A -85,B 0,C 180,E1 -23783.407,E2 -23783.407} C_VEL
LIN {X 0,Y 335.574,Z 576.761,A -85,B 0,C 180,E1 -23785.334,E2 -23785.334} C_VEL
LIN {X 0,Y 340.163,Z 568.153,A -85,B 0,C 180,E1 -23786.937,E2 -23786.937} C_VEL
LIN {X 0,Y 345.024,Z 557.964,A -85,B 0,C 180,E1 -23788.495,E2 -23788.495} C_VEL
LIN {X 0,Y 349.487,Z 547.16,A -85,B 0,C 180,E1 -23789.844,E2 -23789.844} C_VEL
LIN {X 0,Y 354.386,Z 533.21,A -85,B 0,C 180,E1 -23791.254,E2 -23791.254} C_VEL
LIN {X 0,Y 358.225,Z 519.91,A -85,B 0,C 180,E1 -23792.347,E2 -23792.347} C_VEL
LIN {X 0,Y 361.513,Z 505.552,A -85,B 0,C 180,E1 -23793.268,E2 -23793.268} C_VEL
LIN {X 0,Y 364.167,Z 491.136,A -85,B 0,C 180,E1 -23793.986,E2 -23793.986} C_VEL
LIN {X 0,Y 368.205,Z 467.414,A -85,B 0,C 180,E1 -23794.907,E2 -23794.907} C_VEL
LIN {X 0,Y 372.198,Z 445.733,A -85,B 0,C 180,E1 -23795.689,E2 -23795.689} C_VEL
LIN {X 0,Y 370.529,Z 442.036,A -85,B 0,C 180,E1 -23797.063,E2 -23797.063} C_VEL
LIN {X 0,Y 369.502,Z 439.618,A -85,B 0,C 180,E1 -23798.163,E2 -23798.163} C_VEL
LIN {X 0,Y 368.197,Z 436.708,A -85,B 0,C 180,E1 -23799.948,E2 -23799.948} C_VEL
LIN {X 0,Y 367.038,Z 435.426,A -85,B 0,C 180,E1 -23802.582,E2 -23802.582} C_VEL
LIN {X 0,Y 367.068,Z 435.448,A -85,B 0,C 180,E1 -23804.457,E2 -23804.457} C_VEL
LIN {X 0,Y 368.152,Z 437.064,A -85,B 0,C 180,E1 -23807.044,E2 -23807.044} C_VEL
LIN {X 0,Y 368.933,Z 439.347,A -85,B 0,C 180,E1 -23808.283,E2 -23808.283} C_VEL
LIN {X 0,Y 368.822,Z 447.913,A -85,B 0,C 180,E1 -23809.743,E2 -23809.743} C_VEL
LIN {X 0,Y 366.9,Z 467.24,A -85,B 0,C 180,E1 -23811.422,E2 -23811.422} C_VEL
LIN {X 0,Y 365.162,Z 484.834,A -85,B 0,C 180,E1 -23812.739,E2 -23812.739} C_VEL
LIN {X 0,Y 363.547,Z 498.406,A -85,B 0,C 180,E1 -23813.514,E2 -23813.514} C_VEL
LIN {X 0,Y 357.753,Z 530.368,A -85,B 0,C 180,E1 -23814.676,E2 -23814.676} C_VEL
LIN {X 0,Y 353.473,Z 547.663,A -85,B 0,C 180,E1 -23815.442,E2 -23815.442} C_VEL
LIN {X 0,Y 348.209,Z 564.275,A -85,B 0,C 180,E1 -23816.414,E2 -23816.414} C_VEL
LIN {X 0,Y 342.668,Z 579.123,A -85,B 0,C 180,E1 -23817.549,E2 -23817.549} C_VEL
LIN {X 0,Y 336.914,Z 592.675,A -85,B 0,C 180,E1 -23818.858,E2 -23818.858} C_VEL
LIN {X 0,Y 331.561,Z 604.006,A -85,B 0,C 180,E1 -23820.234,E2 -23820.234} C_VEL
LIN {X 0,Y 326.262,Z 614.592,A -85,B 0,C 180,E1 -23821.815,E2 -23821.815} C_VEL
LIN {X 0,Y 321.005,Z 624.334,A -85,B 0,C 180,E1 -23823.63,E2 -23823.63} C_VEL
LIN {X 0,Y 315.818,Z 633.544,A -85,B 0,C 180,E1 -23825.776,E2 -23825.776} C_VEL
LIN {X 0,Y 312.181,Z 639.828,A -85,B 0,C 180,E1 -23827.577,E2 -23827.577} C_VEL
LIN {X 0,Y 307.966,Z 646.718,A -85,B 0,C 180,E1 -23830.052,E2 -23830.052} C_VEL
LIN {X 0,Y 304.807,Z 652.115,A -85,B 0,C 180,E1 -23832.618,E2 -23832.618} C_VEL
LIN {X 0,Y 302.653,Z 656.163,A -85,B 0,C 180,E1 -23835.251,E2 -23835.251} C_VEL
LIN {X 0,Y 301.328,Z 658.922,A -85,B 0,C 180,E1 -23837.924,E2 -23837.924} C_VEL
LIN {X 0,Y 301.074,Z 660.058,A -85,B 0,C 180,E1 -23839.443,E2 -23839.443} C_VEL
LIN {X 0,Y 301.083,Z 661.12,A -85,B 0,C 180,E1 -23839.994,E2 -23839.994} C_VEL
LIN {X 0,Y 300.637,Z 670.837,A -85,B 0,C 180,E1 -23841.964,E2 -23841.964} C_VEL
LIN {X 0,Y 300.43,Z 679.078,A -85,B 0,C 180,E1 -23843.977,E2 -23843.977} C_VEL
LIN {X 0,Y 300.3,Z 685.895,A -85,B 0,C 180,E1 -23845.987,E2 -23845.987} C_VEL
LIN {X 0,Y 300.17,Z 691.49,A -85,B 0,C 180,E1 -23847.994,E2 -23847.994} C_VEL
LIN {X 0,Y 300.124,Z 696.017,A -85,B 0,C 180,E1 -23850,E2 -23850} C_VEL
LIN {X 0,Y 299.923,Z 700.513,A -85,B 0,C 180,E1 -23852.677,E2 -23852.677} C_VEL
LIN {X 0,Y 300.025,Z 703.513,A -85,B 0,C 180,E1 -23855.358,E2 -23855.358} C_VEL
LIN {X 0,Y 300.633,Z 705.152,A -85,B 0,C 180,E1 -23858.036,E2 -23858.036} C_VEL
LIN {X 0,Y 301.904,Z 705.464,A -85,B 0,C 180,E1 -23860.696,E2 -23860.696} C_VEL
LIN {X 0,Y 303.93,Z 704.457,A -85,B 0,C 180,E1 -23863.324,E2 -23863.324} C_VEL
LIN {X 0,Y 306.825,Z 702.119,A -85,B 0,C 180,E1 -23865.899,E2 -23865.899} C_VEL
LIN {X 0,Y 310.055,Z 698.459,A -85,B 0,C 180,E1 -23868.438,E2 -23868.438} C_VEL
LIN {X 0,Y 314.219,Z 693.34,A -85,B 0,C 180,E1 -23870.895,E2 -23870.895} C_VEL
LIN {X 0,Y 317.852,Z 688.442,A -85,B 0,C 180,E1 -23872.684,E2 -23872.684} C_VEL
LIN {X 0,Y 322.475,Z 681.565,A -85,B 0,C 180,E1 -23874.716,E2 -23874.716} C_VEL
LIN {X 0,Y 327.702,Z 673.174,A -85,B 0,C 180,E1 -23876.671,E2 -23876.671} C_VEL
LIN {X 0,Y 333.344,Z 663.087,A -85,B 0,C 180,E1 -23878.557,E2 -23878.557} C_VEL
LIN {X 0,Y 338.614,Z 652.693,A -85,B 0,C 180,E1 -23880.108,E2 -23880.108} C_VEL
LIN {X 0,Y 344.251,Z 640.332,A -85,B 0,C 180,E1 -23881.596,E2 -23881.596} C_VEL
LIN {X 0,Y 349.828,Z 626.588,A -85,B 0,C 180,E1 -23882.896,E2 -23882.896} C_VEL
LIN {X 0,Y 353.998,Z 614.769,A -85,B 0,C 180,E1 -23883.782,E2 -23883.782} C_VEL
LIN {X 0,Y 358.017,Z 601.682,A -85,B 0,C 180,E1 -23884.567,E2 -23884.567} C_VEL
LIN {X 0,Y 362.122,Z 585.441,A -85,B 0,C 180,E1 -23885.306,E2 -23885.306} C_VEL
LIN {X 0,Y 378.73,Z 500.637,A -85,B 0,C 180,E1 -23888.329,E2 -23888.329} C_VEL
LIN {X 0,Y 380.958,Z 485.576,A -85,B 0,C 180,E1 -23889.379,E2 -23889.379} C_VEL
LIN {X 0,Y 382.313,Z 475.839,A -85,B 0,C 180,E1 -23890.214,E2 -23890.214} C_VEL
LIN {X 0,Y 380.752,Z 474.503,A -85,B 0,C 180,E1 -23892.033,E2 -23892.033} C_VEL
LIN {X 0,Y 379.622,Z 474.664,A -85,B 0,C 180,E1 -23894.356,E2 -23894.356} C_VEL
LIN {X 0,Y 379.317,Z 476.264,A -85,B 0,C 180,E1 -23896.069,E2 -23896.069} C_VEL
LIN {X 0,Y 379.492,Z 479.058,A -85,B 0,C 180,E1 -23897.753,E2 -23897.753} C_VEL
LIN {X 0,Y 379.938,Z 483.278,A -85,B 0,C 180,E1 -23899.336,E2 -23899.336} C_VEL
LIN {X 0,Y 378.257,Z 498.933,A -85,B 0,C 180,E1 -23901.054,E2 -23901.054} C_VEL
LIN {X 0,Y 377.308,Z 508.303,A -85,B 0,C 180,E1 -23901.909,E2 -23901.909} C_VEL
LIN {X 0,Y 362.31,Z 585.353,A -85,B 0,C 180,E1 -23904.646,E2 -23904.646} C_VEL
LIN {X 0,Y 358.701,Z 599.581,A -85,B 0,C 180,E1 -23905.295,E2 -23905.295} C_VEL
LIN {X 0,Y 354.136,Z 614.51,A -85,B 0,C 180,E1 -23906.201,E2 -23906.201} C_VEL
LIN {X 0,Y 349.965,Z 626.339,A -85,B 0,C 180,E1 -23907.119,E2 -23907.119} C_VEL
LIN {X 0,Y 344.416,Z 639.893,A -85,B 0,C 180,E1 -23908.421,E2 -23908.421} C_VEL
LIN {X 0,Y 338.838,Z 652.088,A -85,B 0,C 180,E1 -23909.915,E2 -23909.915} C_VEL
LIN {X 0,Y 333.624,Z 662.364,A -85,B 0,C 180,E1 -23911.469,E2 -23911.469} C_VEL
LIN {X 0,Y 327.938,Z 672.402,A -85,B 0,C 180,E1 -23913.35,E2 -23913.35} C_VEL
LIN {X 0,Y 322.08,Z 681.764,A -85,B 0,C 180,E1 -23915.594,E2 -23915.594} C_VEL
LIN {X 0,Y 318.122,Z 687.534,A -85,B 0,C 180,E1 -23917.337,E2 -23917.337} C_VEL
LIN {X 0,Y 313.466,Z 693.767,A -85,B 0,C 180,E1 -23919.736,E2 -23919.736} C_VEL
LIN {X 0,Y 310.342,Z 697.468,A -85,B 0,C 180,E1 -23921.58,E2 -23921.58} C_VEL
LIN {X 0,Y 307.103,Z 701.09,A -85,B 0,C 180,E1 -23924.116,E2 -23924.116} C_VEL
LIN {X 0,Y 304.173,Z 703.401,A -85,B 0,C 180,E1 -23926.687,E2 -23926.687} C_VEL
LIN {X 0,Y 302.06,Z 704.387,A -85,B 0,C 180,E1 -23929.309,E2 -23929.309} C_VEL
LIN {X 0,Y 300.713,Z 704.058,A -85,B 0,C 180,E1 -23931.967,E2 -23931.967} C_VEL
LIN {X 0,Y 300.033,Z 702.41,A -85,B 0,C 180,E1 -23934.642,E2 -23934.642} C_VEL
LIN {X 0,Y 299.814,Z 699.401,A -85,B 0,C 180,E1 -23937.322,E2 -23937.322} C_VEL
LIN {X 0,Y 299.939,Z 694.918,A -85,B 0,C 180,E1 -23940,E2 -23940} C_VEL
LIN {X 0,Y 300.073,Z 690.439,A -85,B 0,C 180,E1 -23942.007,E2 -23942.007} C_VEL
LIN {X 0,Y 300.276,Z 683.882,A -85,B 0,C 180,E1 -23944.348,E2 -23944.348} C_VEL
LIN {X 0,Y 300.466,Z 675.672,A -85,B 0,C 180,E1 -23946.694,E2 -23946.694} C_VEL
LIN {X 0,Y 300.814,Z 667.071,A -85,B 0,C 180,E1 -23948.706,E2 -23948.706} C_VEL
LIN {X 0,Y 301.355,Z 656.652,A -85,B 0,C 180,E1 -23950.717,E2 -23950.717} C_VEL
LIN {X 0,Y 302.144,Z 644.76,A -85,B 0,C 180,E1 -23952.615,E2 -23952.615} C_VEL
LIN {X 0,Y 302.849,Z 632.538,A -85,B 0,C 180,E1 -23954.225,E2 -23954.225} C_VEL
LIN {X 0,Y 303.797,Z 618.578,A -85,B 0,C 180,E1 -23955.719,E2 -23955.719} C_VEL
LIN {X 0,Y 304.634,Z 603.945,A -85,B 0,C 180,E1 -23956.962,E2 -23956.962} C_VEL
LIN {X 0,Y 305.356,Z 588.552,A -85,B 0,C 180,E1 -23957.953,E2 -23957.953} C_VEL
LIN {X 0,Y 306.066,Z 571.498,A -85,B 0,C 180,E1 -23958.731,E2 -23958.731} C_VEL
LIN {X 0,Y 309.418,Z 477.824,A -85,B 0,C 180,E1 -23962.32,E2 -23962.32} C_VEL
LIN {X 0,Y 307.171,Z 449.526,A -85,B 0,C 180,E1 -23963.453,E2 -23963.453} C_VEL
LIN {X 0,Y 306.907,Z 439.617,A -85,B 0,C 180,E1 -23963.853,E2 -23963.853} C_VEL
LIN {X 0,Y 309.519,Z 412.591,A -85,B 0,C 180,E1 -23968.187,E2 -23968.187} C_VEL
LIN {X 0,Y 310.96,Z 398.447,A -85,B 0,C 180,E1 -23970.448,E2 -23970.448} C_VEL
LIN {X 0,Y 307.123,Z 380.516,A -85,B 0,C 180,E1 -23973.593,E2 -23973.593} C_VEL
LIN {X 0,Y 302.614,Z 360.351,A -85,B 0,C 180,E1 -23977.243,E2 -23977.243} C_VEL
LIN {X 0,Y 302.541,Z 360.351,A -85,B 0,C 180,E1 -23980.411,E2 -23980.411} C_VEL
LIN {X 0,Y 302.555,Z 360.353,A -85,B 0,C 180,E1 -23984.137,E2 -23984.137} C_VEL
LIN {X 0,Y 302.559,Z 360.353,A -85,B 0,C 180,E1 -23987.827,E2 -23987.827} C_VEL
LIN {X 0,Y 302.555,Z 360.354,A -85,B 0,C 180,E1 -23991.919,E2 -23991.919} C_VEL
LIN {X 0,Y 302.558,Z 360.352,A -85,B 0,C 180,E1 -23994.636,E2 -23994.636} C_VEL
LIN {X 0,Y 302.534,Z 360.339,A -85,B 0,C 180,E1 -23997.825,E2 -23997.825} C_VEL
LIN {X 0,Y 302.582,Z 360.35,A -85,B 0,C 180,E1 -24001.602,E2 -24001.602} C_VEL
LIN {X 0,Y 302.637,Z 360.346,A -85,B 0,C 180,E1 -24005.014,E2 -24005.014} C_VEL
LIN {X 0,Y 303.621,Z 363.157,A -85,B 0,C 180,E1 -24005.211,E2 -24005.211} C_VEL
LIN {X 0,Y 312.066,Z 380.042,A -85,B 0,C 180,E1 -24006.474,E2 -24006.474} C_VEL
LIN {X 0,Y 318.787,Z 395.389,A -85,B 0,C 180,E1 -24007.469,E2 -24007.469} C_VEL
LIN {X 0,Y 320.12,Z 398.611,A -85,B 0,C 180,E1 -24007.665,E2 -24007.665} C_VEL
LIN {X 0,Y 318.383,Z 462.94,A -85,B 0,C 180,E1 -24009.087,E2 -24009.087} C_VEL
LIN {X 0,Y 318.151,Z 480.029,A -85,B 0,C 180,E1 -24009.543,E2 -24009.543} C_VEL
LIN {X 0,Y 317.519,Z 494.571,A -85,B 0,C 180,E1 -24010.174,E2 -24010.174} C_VEL
LIN {X 0,Y 316.476,Z 508.407,A -85,B 0,C 180,E1 -24011.03,E2 -24011.03} C_VEL
LIN {X 0,Y 315.201,Z 520.796,A -85,B 0,C 180,E1 -24012.041,E2 -24012.041} C_VEL
LIN {X 0,Y 313.842,Z 532.896,A -85,B 0,C 180,E1 -24013.301,E2 -24013.301} C_VEL
LIN {X 0,Y 312.35,Z 543.543,A -85,B 0,C 180,E1 -24014.656,E2 -24014.656} C_VEL
LIN {X 0,Y 310.509,Z 554.255,A -85,B 0,C 180,E1 -24016.299,E2 -24016.299} C_VEL
LIN {X 0,Y 308.55,Z 564.469,A -85,B 0,C 180,E1 -24018.211,E2 -24018.211} C_VEL
LIN {X 0,Y 306.924,Z 572.886,A -85,B 0,C 180,E1 -24020.145,E2 -24020.145} C_VEL
LIN {X 0,Y 305.335,Z 580.956,A -85,B 0,C 180,E1 -24022.42,E2 -24022.42} C_VEL
LIN {X 0,Y 303.997,Z 587.463,A -85,B 0,C 180,E1 -24024.712,E2 -24024.712} C_VEL
LIN {X 0,Y 302.95,Z 593.236,A -85,B 0,C 180,E1 -24027.35,E2 -24027.35} C_VEL
LIN {X 0,Y 302.257,Z 597.483,A -85,B 0,C 180,E1 -24030,E2 -24030} C_VEL
LIN {X 0,Y 301.888,Z 600.338,A -85,B 0,C 180,E1 -24032.66,E2 -24032.66} C_VEL
LIN {X 0,Y 301.958,Z 601.862,A -85,B 0,C 180,E1 -24035.324,E2 -24035.324} C_VEL
LIN {X 0,Y 302.283,Z 602.106,A -85,B 0,C 180,E1 -24037.992,E2 -24037.992} C_VEL
LIN {X 0,Y 302.941,Z 601.061,A -85,B 0,C 180,E1 -24040.66,E2 -24040.66} C_VEL
LIN {X 0,Y 304.08,Z 598.686,A -85,B 0,C 180,E1 -24043.318,E2 -24043.318} C_VEL
LIN {X 0,Y 305.652,Z 594.893,A -85,B 0,C 180,E1 -24045.962,E2 -24045.962} C_VEL
LIN {X 0,Y 307.606,Z 589.542,A -85,B 0,C 180,E1 -24048.59,E2 -24048.59} C_VEL
LIN {X 0,Y 309.383,Z 584.451,A -85,B 0,C 180,E1 -24050.544,E2 -24050.544} C_VEL
LIN {X 0,Y 311.445,Z 578.219,A -85,B 0,C 180,E1 -24052.479,E2 -24052.479} C_VEL
LIN {X 0,Y 314.124,Z 569.337,A -85,B 0,C 180,E1 -24054.715,E2 -24054.715} C_VEL
LIN {X 0,Y 316.731,Z 559.975,A -85,B 0,C 180,E1 -24056.605,E2 -24056.605} C_VEL
LIN {X 0,Y 319.219,Z 549.759,A -85,B 0,C 180,E1 -24058.296,E2 -24058.296} C_VEL
LIN {X 0,Y 321.439,Z 539.322,A -85,B 0,C 180,E1 -24059.719,E2 -24059.719} C_VEL
LIN {X 0,Y 323.843,Z 526.74,A -85,B 0,C 180,E1 -24061.091,E2 -24061.091} C_VEL
LIN {X 0,Y 325.514,Z 514.468,A -85,B 0,C 180,E1 -24062.18,E2 -24062.18} C_VEL
LIN {X 0,Y 326.953,Z 501.301,A -85,B 0,C 180,E1 -24063.079,E2 -24063.079} C_VEL
LIN {X 0,Y 328.003,Z 487.663,A -85,B 0,C 180,E1 -24063.762,E2 -24063.762} C_VEL
LIN {X 0,Y 328.484,Z 473.772,A -85,B 0,C 180,E1 -24064.235,E2 -24064.235} C_VEL
LIN {X 0,Y 330.606,Z 411.423,A -85,B 0,C 180,E1 -24065.589,E2 -24065.589} C_VEL
LIN {X 0,Y 322.823,Z 395.748,A -85,B 0,C 180,E1 -24066.925,E2 -24066.925} C_VEL
LIN {X 0,Y 313.739,Z 379.324,A -85,B 0,C 180,E1 -24068.546,E2 -24068.546} C_VEL
LIN {X 0,Y 306.598,Z 367.898,A -85,B 0,C 180,E1 -24069.872,E2 -24069.872} C_VEL
LIN {X 0,Y 304.441,Z 364.42,A -85,B 0,C 180,E1 -24070.29,E2 -24070.29} C_VEL
LIN {X 0,Y 302.938,Z 362.113,A -85,B 0,C 180,E1 -24070.583,E2 -24070.583} C_VEL
LIN {X 0,Y 302.516,Z 360.364,A -85,B 0,C 180,E1 -24070.726,E2 -24070.726} C_VEL
LIN {X 0,Y 302.518,Z 360.359,A -85,B 0,C 180,E1 -24074.129,E2 -24074.129} C_VEL
LIN {X 0,Y 302.524,Z 360.352,A -85,B 0,C 180,E1 -24077.821,E2 -24077.821} C_VEL
LIN {X 0,Y 302.504,Z 360.322,A -85,B 0,C 180,E1 -24081.931,E2 -24081.931} C_VEL
LIN {X 0,Y 302.537,Z 360.316,A -85,B 0,C 180,E1 -24084.633,E2 -24084.633} C_VEL
LIN {X 0,Y 302.516,Z 360.355,A -85,B 0,C 180,E1 -24087.822,E2 -24087.822} C_VEL
LIN {X 0,Y 302.566,Z 360.353,A -85,B 0,C 180,E1 -24091.608,E2 -24091.608} C_VEL
LIN {X 0,Y 302.562,Z 360.346,A -85,B 0,C 180,E1 -24095.373,E2 -24095.373} C_VEL
LIN {X 0,Y 302.65,Z 360.343,A -85,B 0,C 180,E1 -24096.559,E2 -24096.559} C_VEL
LIN {X 0,Y 307.745,Z 380.953,A -85,B 0,C 180,E1 -24097.464,E2 -24097.464} C_VEL
LIN {X 0,Y 308.592,Z 384.007,A -85,B 0,C 180,E1 -24097.596,E2 -24097.596} C_VEL
LIN {X 0,Y 306.552,Z 447.09,A -85,B 0,C 180,E1 -24099.933,E2 -24099.933} C_VEL
LIN {X 0,Y 305.826,Z 452.853,A -85,B 0,C 180,E1 -24100.14,E2 -24100.14} C_VEL
LIN {X 0,Y 299.589,Z 471.388,A -85,B 0,C 180,E1 -24100.812,E2 -24100.812} C_VEL
LIN {X 0,Y 298.927,Z 477.107,A -85,B 0,C 180,E1 -24101.063,E2 -24101.063} C_VEL
LIN {X 0,Y 298.369,Z 491.945,A -85,B 0,C 180,E1 -24101.877,E2 -24101.877} C_VEL
LIN {X 0,Y 297.723,Z 507.144,A -85,B 0,C 180,E1 -24102.985,E2 -24102.985} C_VEL
LIN {X 0,Y 296.997,Z 520.854,A -85,B 0,C 180,E1 -24104.263,E2 -24104.263} C_VEL
LIN {X 0,Y 296.301,Z 534.466,A -85,B 0,C 180,E1 -24105.827,E2 -24105.827} C_VEL
LIN {X 0,Y 295.654,Z 546.609,A -85,B 0,C 180,E1 -24107.515,E2 -24107.515} C_VEL
LIN {X 0,Y 294.979,Z 557.832,A -85,B 0,C 180,E1 -24109.395,E2 -24109.395} C_VEL
LIN {X 0,Y 294.484,Z 568.078,A -85,B 0,C 180,E1 -24111.45,E2 -24111.45} C_VEL
LIN {X 0,Y 294.134,Z 578.029,A -85,B 0,C 180,E1 -24113.848,E2 -24113.848} C_VEL
LIN {X 0,Y 294.109,Z 586.152,A -85,B 0,C 180,E1 -24116.244,E2 -24116.244} C_VEL
LIN {X 0,Y 294.272,Z 592.727,A -85,B 0,C 180,E1 -24118.636,E2 -24118.636} C_VEL
LIN {X 0,Y 294.847,Z 598.635,A -85,B 0,C 180,E1 -24121.361,E2 -24121.361} C_VEL
LIN {X 0,Y 295.924,Z 603.02,A -85,B 0,C 180,E1 -24124.072,E2 -24124.072} C_VEL
LIN {X 0,Y 297.585,Z 605.973,A -85,B 0,C 180,E1 -24126.758,E2 -24126.758} C_VEL
LIN {X 0,Y 299.655,Z 607.547,A -85,B 0,C 180,E1 -24129.417,E2 -24129.417} C_VEL
LIN {X 0,Y 302.405,Z 607.739,A -85,B 0,C 180,E1 -24132.032,E2 -24132.032} C_VEL
LIN {X 0,Y 306.112,Z 606.495,A -85,B 0,C 180,E1 -24134.578,E2 -24134.578} C_VEL
LIN {X 0,Y 310.179,Z 603.902,A -85,B 0,C 180,E1 -24137.071,E2 -24137.071} C_VEL
LIN {X 0,Y 314.671,Z 599.928,A -85,B 0,C 180,E1 -24139.505,E2 -24139.505} C_VEL
LIN {X 0,Y 318.435,Z 595.852,A -85,B 0,C 180,E1 -24141.281,E2 -24141.281} C_VEL
LIN {X 0,Y 323.87,Z 589.057,A -85,B 0,C 180,E1 -24143.584,E2 -24143.584} C_VEL
LIN {X 0,Y 328.941,Z 581.51,A -85,B 0,C 180,E1 -24145.544,E2 -24145.544} C_VEL
LIN {X 0,Y 334.477,Z 572.263,A -85,B 0,C 180,E1 -24147.433,E2 -24147.433} C_VEL
LIN {X 0,Y 339.499,Z 562.668,A -85,B 0,C 180,E1 -24149.002,E2 -24149.002} C_VEL
LIN {X 0,Y 345.179,Z 550.113,A -85,B 0,C 180,E1 -24150.653,E2 -24150.653} C_VEL
LIN {X 0,Y 350.131,Z 537.197,A -85,B 0,C 180,E1 -24152.015,E2 -24152.015} C_VEL
LIN {X 0,Y 354.507,Z 523.23,A -85,B 0,C 180,E1 -24153.204,E2 -24153.204} C_VEL
LIN {X 0,Y 357.959,Z 509.943,A -85,B 0,C 180,E1 -24154.107,E2 -24154.107} C_VEL
LIN {X 0,Y 360.855,Z 495.562,A -85,B 0,C 180,E1 -24154.853,E2 -24154.853} C_VEL
LIN {X 0,Y 365.181,Z 471.402,A -85,B 0,C 180,E1 -24155.834,E2 -24155.834} C_VEL
LIN {X 0,Y 369.222,Z 450.584,A -85,B 0,C 180,E1 -24156.571,E2 -24156.571} C_VEL
LIN {X 0,Y 367.694,Z 446.618,A -85,B 0,C 180,E1 -24158.177,E2 -24158.177} C_VEL
LIN {X 0,Y 366.324,Z 443.491,A -85,B 0,C 180,E1 -24160.107,E2 -24160.107} C_VEL
LIN {X 0,Y 365.363,Z 442.386,A -85,B 0,C 180,E1 -24162.143,E2 -24162.143} C_VEL
LIN {X 0,Y 365.318,Z 442.333,A -85,B 0,C 180,E1 -24164.444,E2 -24164.444} C_VEL
LIN {X 0,Y 366.262,Z 443.798,A -85,B 0,C 180,E1 -24166.832,E2 -24166.832} C_VEL
LIN {X 0,Y 366.719,Z 445.65,A -85,B 0,C 180,E1 -24167.785,E2 -24167.785} C_VEL
LIN {X 0,Y 366.42,Z 452.337,A -85,B 0,C 180,E1 -24168.935,E2 -24168.935} C_VEL
LIN {X 0,Y 364.148,Z 471.481,A -85,B 0,C 180,E1 -24170.597,E2 -24170.597} C_VEL
LIN {X 0,Y 362.258,Z 488.357,A -85,B 0,C 180,E1 -24171.861,E2 -24171.861} C_VEL
LIN {X 0,Y 360.766,Z 499.159,A -85,B 0,C 180,E1 -24172.49,E2 -24172.49} C_VEL
LIN {X 0,Y 354.9,Z 529.924,A -85,B 0,C 180,E1 -24173.606,E2 -24173.606} C_VEL
LIN {X 0,Y 350.655,Z 546.153,A -85,B 0,C 180,E1 -24174.336,E2 -24174.336} C_VEL
LIN {X 0,Y 344.855,Z 563.563,A -85,B 0,C 180,E1 -24175.339,E2 -24175.339} C_VEL
LIN {X 0,Y 339.658,Z 576.942,A -85,B 0,C 180,E1 -24176.343,E2 -24176.343} C_VEL
LIN {X 0,Y 333.616,Z 590.475,A -85,B 0,C 180,E1 -24177.63,E2 -24177.63} C_VEL
LIN {X 0,Y 327.526,Z 602.935,A -85,B 0,C 180,E1 -24179.118,E2 -24179.118} C_VEL
LIN {X 0,Y 321.89,Z 613.402,A -85,B 0,C 180,E1 -24180.685,E2 -24180.685} C_VEL
LIN {X 0,Y 315.959,Z 623.775,A -85,B 0,C 180,E1 -24182.641,E2 -24182.641} C_VEL
LIN {X 0,Y 310.793,Z 632.274,A -85,B 0,C 180,E1 -24184.646,E2 -24184.646} C_VEL
LIN {X 0,Y 305.666,Z 640.403,A -85,B 0,C 180,E1 -24187.073,E2 -24187.073} C_VEL
LIN {X 0,Y 301.304,Z 646.921,A -85,B 0,C 180,E1 -24189.591,E2 -24189.591} C_VEL
LIN {X 0,Y 298,Z 652.005,A -85,B 0,C 180,E1 -24192.208,E2 -24192.208} C_VEL
LIN {X 0,Y 295.741,Z 655.744,A -85,B 0,C 180,E1 -24194.898,E2 -24194.898} C_VEL
LIN {X 0,Y 294.329,Z 658.231,A -85,B 0,C 180,E1 -24197.632,E2 -24197.632} C_VEL
LIN {X 0,Y 294.073,Z 659.083,A -85,B 0,C 180,E1 -24199.015,E2 -24199.015} C_VEL
LIN {X 0,Y 294.045,Z 661.105,A -85,B 0,C 180,E1 -24200.228,E2 -24200.228} C_VEL
LIN {X 0,Y 293.608,Z 670.214,A -85,B 0,C 180,E1 -24202.115,E2 -24202.115} C_VEL
LIN {X 0,Y 293.416,Z 678.561,A -85,B 0,C 180,E1 -24204.177,E2 -24204.177} C_VEL
LIN {X 0,Y 293.276,Z 685.425,A -85,B 0,C 180,E1 -24206.234,E2 -24206.234} C_VEL
LIN {X 0,Y 293.174,Z 691.906,A -85,B 0,C 180,E1 -24208.631,E2 -24208.631} C_VEL
LIN {X 0,Y 292.998,Z 696.299,A -85,B 0,C 180,E1 -24210.685,E2 -24210.685} C_VEL
LIN {X 0,Y 292.889,Z 699.745,A -85,B 0,C 180,E1 -24212.741,E2 -24212.741} C_VEL
LIN {X 0,Y 292.987,Z 703.027,A -85,B 0,C 180,E1 -24215.487,E2 -24215.487} C_VEL
LIN {X 0,Y 293.59,Z 704.928,A -85,B 0,C 180,E1 -24218.23,E2 -24218.23} C_VEL
LIN {X 0,Y 294.932,Z 705.514,A -85,B 0,C 180,E1 -24220.952,E2 -24220.952} C_VEL
LIN {X 0,Y 297.029,Z 704.795,A -85,B 0,C 180,E1 -24223.64,E2 -24223.64} C_VEL
LIN {X 0,Y 300.025,Z 702.754,A -85,B 0,C 180,E1 -24226.269,E2 -24226.269} C_VEL
LIN {X 0,Y 303.393,Z 699.413,A -85,B 0,C 180,E1 -24228.858,E2 -24228.858} C_VEL
LIN {X 0,Y 306.553,Z 695.991,A -85,B 0,C 180,E1 -24230.742,E2 -24230.742} C_VEL
LIN {X 0,Y 311.493,Z 690.108,A -85,B 0,C 180,E1 -24233.173,E2 -24233.173} C_VEL
LIN {X 0,Y 316.986,Z 682.577,A -85,B 0,C 180,E1 -24235.524,E2 -24235.524} C_VEL
LIN {X 0,Y 322.462,Z 674.428,A -85,B 0,C 180,E1 -24237.49,E2 -24237.49} C_VEL
LIN {X 0,Y 328.35,Z 664.647,A -85,B 0,C 180,E1 -24239.383,E2 -24239.383} C_VEL
LIN {X 0,Y 333.831,Z 654.665,A -85,B 0,C 180,E1 -24240.934,E2 -24240.934} C_VEL
LIN {X 0,Y 339.676,Z 642.793,A -85,B 0,C 180,E1 -24242.422,E2 -24242.422} C_VEL
LIN {X 0,Y 344.889,Z 630.921,A -85,B 0,C 180,E1 -24243.602,E2 -24243.602} C_VEL
LIN {X 0,Y 349.467,Z 619.15,A -85,B 0,C 180,E1 -24244.555,E2 -24244.555} C_VEL
LIN {X 0,Y 354.674,Z 603.717,A -85,B 0,C 180,E1 -24245.524,E2 -24245.524} C_VEL
LIN {X 0,Y 358.641,Z 589.226,A -85,B 0,C 180,E1 -24246.214,E2 -24246.214} C_VEL
LIN {X 0,Y 363.44,Z 566.299,A -85,B 0,C 180,E1 -24247.076,E2 -24247.076} C_VEL
LIN {X 0,Y 376.611,Z 502.398,A -85,B 0,C 180,E1 -24249.321,E2 -24249.321} C_VEL
LIN {X 0,Y 378.98,Z 488.016,A -85,B 0,C 180,E1 -24250.342,E2 -24250.342} C_VEL
LIN {X 0,Y 379.904,Z 482.123,A -85,B 0,C 180,E1 -24250.86,E2 -24250.86} C_VEL
LIN {X 0,Y 378.81,Z 481.32,A -85,B 0,C 180,E1 -24252.301,E2 -24252.301} C_VEL
LIN {X 0,Y 377.837,Z 481.606,A -85,B 0,C 180,E1 -24254.395,E2 -24254.395} C_VEL
LIN {X 0,Y 377.509,Z 483.255,A -85,B 0,C 180,E1 -24256.038,E2 -24256.038} C_VEL
LIN {X 0,Y 377.595,Z 485.66,A -85,B 0,C 180,E1 -24257.482,E2 -24257.482} C_VEL
LIN {X 0,Y 377.773,Z 488.854,A -85,B 0,C 180,E1 -24258.69,E2 -24258.69} C_VEL
LIN {X 0,Y 375.806,Z 504.129,A -85,B 0,C 180,E1 -24260.348,E2 -24260.348} C_VEL
LIN {X 0,Y 374.971,Z 510.646,A -85,B 0,C 180,E1 -24260.934,E2 -24260.934} C_VEL
LIN {X 0,Y 359.489,Z 586.321,A -85,B 0,C 180,E1 -24263.626,E2 -24263.626} C_VEL
LIN {X 0,Y 355.735,Z 600.362,A -85,B 0,C 180,E1 -24264.271,E2 -24264.271} C_VEL
LIN {X 0,Y 350.995,Z 615.062,A -85,B 0,C 180,E1 -24265.164,E2 -24265.164} C_VEL
LIN {X 0,Y 346.63,Z 626.754,A -85,B 0,C 180,E1 -24266.067,E2 -24266.067} C_VEL
LIN {X 0,Y 340.855,Z 640.139,A -85,B 0,C 180,E1 -24267.355,E2 -24267.355} C_VEL
LIN {X 0,Y 335.025,Z 652.227,A -85,B 0,C 180,E1 -24268.839,E2 -24268.839} C_VEL
LIN {X 0,Y 329.546,Z 662.425,A -85,B 0,C 180,E1 -24270.385,E2 -24270.385} C_VEL
LIN {X 0,Y 323.522,Z 672.42,A -85,B 0,C 180,E1 -24272.258,E2 -24272.258} C_VEL
LIN {X 0,Y 317.293,Z 681.745,A -85,B 0,C 180,E1 -24274.503,E2 -24274.503} C_VEL
LIN {X 0,Y 311.78,Z 689.229,A -85,B 0,C 180,E1 -24276.849,E2 -24276.849} C_VEL
LIN {X 0,Y 306.941,Z 695.053,A -85,B 0,C 180,E1 -24279.286,E2 -24279.286} C_VEL
LIN {X 0,Y 303.705,Z 698.451,A -85,B 0,C 180,E1 -24281.163,E2 -24281.163} C_VEL
LIN {X 0,Y 300.306,Z 701.76,A -85,B 0,C 180,E1 -24283.747,E2 -24283.747} C_VEL
LIN {X 0,Y 297.273,Z 703.775,A -85,B 0,C 180,E1 -24286.372,E2 -24286.372} C_VEL
LIN {X 0,Y 295.083,Z 704.475,A -85,B 0,C 180,E1 -24289.054,E2 -24289.054} C_VEL
LIN {X 0,Y 293.671,Z 703.874,A -85,B 0,C 180,E1 -24291.773,E2 -24291.773} C_VEL
LIN {X 0,Y 292.996,Z 701.964,A -85,B 0,C 180,E1 -24294.513,E2 -24294.513} C_VEL
LIN {X 0,Y 292.766,Z 698.679,A -85,B 0,C 180,E1 -24297.258,E2 -24297.258} C_VEL
LIN {X 0,Y 292.907,Z 693.899,A -85,B 0,C 180,E1 -24300,E2 -24300} C_VEL
LIN {X 0,Y 293.054,Z 689.228,A -85,B 0,C 180,E1 -24302.055,E2 -24302.055} C_VEL
LIN {X 0,Y 293.272,Z 682.377,A -85,B 0,C 180,E1 -24304.452,E2 -24304.452} C_VEL
LIN {X 0,Y 293.477,Z 673.781,A -85,B 0,C 180,E1 -24306.854,E2 -24306.854} C_VEL
LIN {X 0,Y 293.884,Z 664.804,A -85,B 0,C 180,E1 -24308.913,E2 -24308.913} C_VEL
LIN {X 0,Y 294.402,Z 653.99,A -85,B 0,C 180,E1 -24310.973,E2 -24310.973} C_VEL
LIN {X 0,Y 295.104,Z 643.781,A -85,B 0,C 180,E1 -24312.6,E2 -24312.6} C_VEL
LIN {X 0,Y 295.819,Z 631.596,A -85,B 0,C 180,E1 -24314.221,E2 -24314.221} C_VEL
LIN {X 0,Y 296.777,Z 617.406,A -85,B 0,C 180,E1 -24315.749,E2 -24315.749} C_VEL
LIN {X 0,Y 297.604,Z 602.514,A -85,B 0,C 180,E1 -24317.022,E2 -24317.022} C_VEL
LIN {X 0,Y 298.325,Z 586.649,A -85,B 0,C 180,E1 -24318.038,E2 -24318.038} C_VEL
LIN {X 0,Y 299.046,Z 569.18,A -85,B 0,C 180,E1 -24318.832,E2 -24318.832} C_VEL
LIN {X 0,Y 302.318,Z 477.827,A -85,B 0,C 180,E1 -24322.448,E2 -24322.448} C_VEL
LIN {X 0,Y 300.125,Z 449.86,A -85,B 0,C 180,E1 -24323.605,E2 -24323.605} C_VEL
LIN {X 0,Y 299.899,Z 439.521,A -85,B 0,C 180,E1 -24324.044,E2 -24324.044} C_VEL
LIN {X 0,Y 302.503,Z 412.985,A -85,B 0,C 180,E1 -24328.371,E2 -24328.371} C_VEL
LIN {X 0,Y 303.877,Z 400.065,A -85,B 0,C 180,E1 -24330.472,E2 -24330.472} C_VEL
LIN {X 0,Y 302.369,Z 391.742,A -85,B 0,C 180,E1 -24331.932,E2 -24331.932} C_VEL
LIN {X 0,Y 297.298,Z 368.808,A -85,B 0,C 180,E1 -24336.087,E2 -24336.087} C_VEL
LIN {X 0,Y 295.568,Z 361.228,A -85,B 0,C 180,E1 -24337.534,E2 -24337.534} C_VEL
LIN {X 0,Y 295.485,Z 361.232,A -85,B 0,C 180,E1 -24341.586,E2 -24341.586} C_VEL
LIN {X 0,Y 295.497,Z 361.227,A -85,B 0,C 180,E1 -24345.327,E2 -24345.327} C_VEL
LIN {X 0,Y 295.498,Z 361.227,A -85,B 0,C 180,E1 -24349.335,E2 -24349.335} C_VEL
LIN {X 0,Y 295.508,Z 361.231,A -85,B 0,C 180,E1 -24351.955,E2 -24351.955} C_VEL
LIN {X 0,Y 295.489,Z 361.234,A -85,B 0,C 180,E1 -24356.065,E2 -24356.065} C_VEL
LIN {X 0,Y 295.507,Z 361.228,A -85,B 0,C 180,E1 -24360.148,E2 -24360.148} C_VEL
LIN {X 0,Y 295.584,Z 361.222,A -85,B 0,C 180,E1 -24364.295,E2 -24364.295} C_VEL
LIN {X 0,Y 296.612,Z 364.09,A -85,B 0,C 180,E1 -24364.503,E2 -24364.503} C_VEL
LIN {X 0,Y 305.259,Z 381.102,A -85,B 0,C 180,E1 -24365.846,E2 -24365.846} C_VEL
LIN {X 0,Y 312.305,Z 396.985,A -85,B 0,C 180,E1 -24366.925,E2 -24366.925} C_VEL
LIN {X 0,Y 313.705,Z 400.363,A -85,B 0,C 180,E1 -24367.138,E2 -24367.138} C_VEL
LIN {X 0,Y 311.928,Z 464.793,A -85,B 0,C 180,E1 -24368.591,E2 -24368.591} C_VEL
LIN {X 0,Y 311.571,Z 482.607,A -85,B 0,C 180,E1 -24369.091,E2 -24369.091} C_VEL
LIN {X 0,Y 310.951,Z 496.536,A -85,B 0,C 180,E1 -24369.737,E2 -24369.737} C_VEL
LIN {X 0,Y 309.905,Z 510.051,A -85,B 0,C 180,E1 -24370.612,E2 -24370.612} C_VEL
LIN {X 0,Y 308.544,Z 522.255,A -85,B 0,C 180,E1 -24371.64,E2 -24371.64} C_VEL
LIN {X 0,Y 307.142,Z 534.22,A -85,B 0,C 180,E1 -24372.925,E2 -24372.925} C_VEL
LIN {X 0,Y 305.365,Z 546.031,A -85,B 0,C 180,E1 -24374.484,E2 -24374.484} C_VEL
LIN {X 0,Y 303.329,Z 557.226,A -85,B 0,C 180,E1 -24376.309,E2 -24376.309} C_VEL
LIN {X 0,Y 301.389,Z 567.012,A -85,B 0,C 180,E1 -24378.267,E2 -24378.267} C_VEL
LIN {X 0,Y 299.549,Z 576.336,A -85,B 0,C 180,E1 -24380.579,E2 -24380.579} C_VEL
LIN {X 0,Y 298.117,Z 582.913,A -85,B 0,C 180,E1 -24382.575,E2 -24382.575} C_VEL
LIN {X 0,Y 296.992,Z 588.386,A -85,B 0,C 180,E1 -24384.587,E2 -24384.587} C_VEL
LIN {X 0,Y 295.924,Z 594.122,A -85,B 0,C 180,E1 -24387.287,E2 -24387.287} C_VEL
LIN {X 0,Y 295.189,Z 598.34,A -85,B 0,C 180,E1 -24390,E2 -24390} C_VEL
LIN {X 0,Y 294.844,Z 601.16,A -85,B 0,C 180,E1 -24392.724,E2 -24392.724} C_VEL
LIN {X 0,Y 294.908,Z 602.656,A -85,B 0,C 180,E1 -24395.452,E2 -24395.452} C_VEL
LIN {X 0,Y 295.259,Z 602.869,A -85,B 0,C 180,E1 -24398.183,E2 -24398.183} C_VEL
LIN {X 0,Y 295.961,Z 601.793,A -85,B 0,C 180,E1 -24400.914,E2 -24400.914} C_VEL
LIN {X 0,Y 297.178,Z 599.382,A -85,B 0,C 180,E1 -24403.633,E2 -24403.633} C_VEL
LIN {X 0,Y 298.827,Z 595.541,A -85,B 0,C 180,E1 -24406.337,E2 -24406.337} C_VEL
LIN {X 0,Y 300.884,Z 590.153,A -85,B 0,C 180,E1 -24409.021,E2 -24409.021} C_VEL
LIN {X 0,Y 302.736,Z 585.025,A -85,B 0,C 180,E1 -24411.016,E2 -24411.016} C_VEL
LIN {X 0,Y 304.878,Z 578.769,A -85,B 0,C 180,E1 -24412.99,E2 -24412.99} C_VEL
LIN {X 0,Y 307.668,Z 569.814,A -85,B 0,C 180,E1 -24415.269,E2 -24415.269} C_VEL
LIN {X 0,Y 310.407,Z 560.391,A -85,B 0,C 180,E1 -24417.191,E2 -24417.191} C_VEL
LIN {X 0,Y 312.97,Z 549.985,A -85,B 0,C 180,E1 -24418.935,E2 -24418.935} C_VEL
LIN {X 0,Y 315.544,Z 538.297,A -85,B 0,C 180,E1 -24420.516,E2 -24420.516} C_VEL
LIN {X 0,Y 317.764,Z 526.885,A -85,B 0,C 180,E1 -24421.754,E2 -24421.754} C_VEL
LIN {X 0,Y 319.5,Z 514.452,A -85,B 0,C 180,E1 -24422.861,E2 -24422.861} C_VEL
LIN {X 0,Y 321.044,Z 500.468,A -85,B 0,C 180,E1 -24423.81,E2 -24423.81} C_VEL
LIN {X 0,Y 322.078,Z 486.399,A -85,B 0,C 180,E1 -24424.498,E2 -24424.498} C_VEL
LIN {X 0,Y 322.552,Z 471.688,A -85,B 0,C 180,E1 -24424.962,E2 -24424.962} C_VEL
LIN {X 0,Y 324.684,Z 413.633,A -85,B 0,C 180,E1 -24426.226,E2 -24426.226} C_VEL
LIN {X 0,Y 316.079,Z 396.564,A -85,B 0,C 180,E1 -24427.759,E2 -24427.759} C_VEL
LIN {X 0,Y 308.038,Z 382.242,A -85,B 0,C 180,E1 -24429.251,E2 -24429.251} C_VEL
LIN {X 0,Y 299.741,Z 368.963,A -85,B 0,C 180,E1 -24430.866,E2 -24430.866} C_VEL
LIN {X 0,Y 297.545,Z 365.424,A -85,B 0,C 180,E1 -24431.315,E2 -24431.315} C_VEL
LIN {X 0,Y 295.879,Z 362.881,A -85,B 0,C 180,E1 -24431.658,E2 -24431.658} C_VEL
LIN {X 0,Y 295.488,Z 361.235,A -85,B 0,C 180,E1 -24431.816,E2 -24431.816} C_VEL
LIN {X 0,Y 295.467,Z 361.234,A -85,B 0,C 180,E1 -24435.332,E2 -24435.332} C_VEL
LIN {X 0,Y 295.463,Z 361.238,A -85,B 0,C 180,E1 -24439.343,E2 -24439.343} C_VEL
LIN {X 0,Y 295.505,Z 361.182,A -85,B 0,C 180,E1 -24443.699,E2 -24443.699} C_VEL
LIN {X 0,Y 295.487,Z 361.232,A -85,B 0,C 180,E1 -24446.96,E2 -24446.96} C_VEL
LIN {X 0,Y 295.492,Z 361.232,A -85,B 0,C 180,E1 -24451.291,E2 -24451.291} C_VEL
LIN {X 0,Y 295.541,Z 361.215,A -85,B 0,C 180,E1 -24454.747,E2 -24454.747} C_VEL
LIN {X 0,Y 295.584,Z 361.224,A -85,B 0,C 180,E1 -24456.429,E2 -24456.429} C_VEL
LIN {X 0,Y 300.62,Z 381.668,A -85,B 0,C 180,E1 -24457.352,E2 -24457.352} C_VEL
LIN {X 0,Y 301.522,Z 385.049,A -85,B 0,C 180,E1 -24457.5,E2 -24457.5} C_VEL
LIN {X 0,Y 298.915,Z 476.321,A -85,B 0,C 180,E1 -24461.026,E2 -24461.026} C_VEL
LIN {X 0,Y 298.927,Z 477.107,A -85,B 0,C 180,E1 -24461.063,E2 -24461.063} C_VEL
LIN {X 0,Y 298.626,Z 480.908,A -85,B 0,C 180,E1 -24461.247,E2 -24461.247} C_VEL
LIN {X 0,Y 296.497,Z 488.238,A -85,B 0,C 180,E1 -24461.645,E2 -24461.645} C_VEL
LIN {X 0,Y 291.625,Z 500.61,A -85,B 0,C 180,E1 -24462.476,E2 -24462.476} C_VEL
LIN {X 0,Y 290.69,Z 506.052,A -85,B 0,C 180,E1 -24462.908,E2 -24462.908} C_VEL
LIN {X 0,Y 289.923,Z 520.315,A -85,B 0,C 180,E1 -24464.228,E2 -24464.228} C_VEL
LIN {X 0,Y 289.212,Z 534.414,A -85,B 0,C 180,E1 -24465.872,E2 -24465.872} C_VEL
LIN {X 0,Y 288.516,Z 547.533,A -85,B 0,C 180,E1 -24467.735,E2 -24467.735} C_VEL
LIN {X 0,Y 287.891,Z 557.814,A -85,B 0,C 180,E1 -24469.486,E2 -24469.486} C_VEL
LIN {X 0,Y 287.37,Z 568.203,A -85,B 0,C 180,E1 -24471.59,E2 -24471.59} C_VEL
LIN {X 0,Y 287.037,Z 578.238,A -85,B 0,C 180,E1 -24474.047,E2 -24474.047} C_VEL
LIN {X 0,Y 287.015,Z 586.511,A -85,B 0,C 180,E1 -24476.502,E2 -24476.502} C_VEL
LIN {X 0,Y 287.221,Z 593.537,A -85,B 0,C 180,E1 -24479.09,E2 -24479.09} C_VEL
LIN {X 0,Y 287.974,Z 599.883,A -85,B 0,C 180,E1 -24482.091,E2 -24482.091} C_VEL
LIN {X 0,Y 288.873,Z 603.251,A -85,B 0,C 180,E1 -24484.171,E2 -24484.171} C_VEL
LIN {X 0,Y 290.555,Z 606.491,A -85,B 0,C 180,E1 -24486.923,E2 -24486.923} C_VEL
LIN {X 0,Y 292.721,Z 608.373,A -85,B 0,C 180,E1 -24489.642,E2 -24489.642} C_VEL
LIN {X 0,Y 295.56,Z 608.906,A -85,B 0,C 180,E1 -24492.315,E2 -24492.315} C_VEL
LIN {X 0,Y 299.402,Z 608.013,A -85,B 0,C 180,E1 -24494.912,E2 -24494.912} C_VEL
LIN {X 0,Y 303.644,Z 605.769,A -85,B 0,C 180,E1 -24497.45,E2 -24497.45} C_VEL
LIN {X 0,Y 308.279,Z 602.101,A -85,B 0,C 180,E1 -24499.926,E2 -24499.926} C_VEL
LIN {X 0,Y 313.589,Z 596.93,A -85,B 0,C 180,E1 -24502.316,E2 -24502.316} C_VEL
LIN {X 0,Y 317.826,Z 591.974,A -85,B 0,C 180,E1 -24504.061,E2 -24504.061} C_VEL
LIN {X 0,Y 323.902,Z 583.834,A -85,B 0,C 180,E1 -24506.315,E2 -24506.315} C_VEL
LIN {X 0,Y 329.669,Z 574.837,A -85,B 0,C 180,E1 -24508.212,E2 -24508.212} C_VEL
LIN {X 0,Y 335.814,Z 563.905,A -85,B 0,C 180,E1 -24510.039,E2 -24510.039} C_VEL
LIN {X 0,Y 341.277,Z 552.473,A -85,B 0,C 180,E1 -24511.558,E2 -24511.558} C_VEL
LIN {X 0,Y 346.951,Z 538.652,A -85,B 0,C 180,E1 -24513.031,E2 -24513.031} C_VEL
LIN {X 0,Y 351.174,Z 526.019,A -85,B 0,C 180,E1 -24514.123,E2 -24514.123} C_VEL
LIN {X 0,Y 355.48,Z 510.303,A -85,B 0,C 180,E1 -24515.194,E2 -24515.194} C_VEL
LIN {X 0,Y 358.536,Z 495.915,A -85,B 0,C 180,E1 -24515.936,E2 -24515.936} C_VEL
LIN {X 0,Y 363.063,Z 471.842,A -85,B 0,C 180,E1 -24516.897,E2 -24516.897} C_VEL
LIN {X 0,Y 366.425,Z 455.384,A -85,B 0,C 180,E1 -24517.487,E2 -24517.487} C_VEL
LIN {X 0,Y 365.27,Z 452.494,A -85,B 0,C 180,E1 -24518.869,E2 -24518.869} C_VEL
LIN {X 0,Y 364.427,Z 450.253,A -85,B 0,C 180,E1 -24520.303,E2 -24520.303} C_VEL
LIN {X 0,Y 363.578,Z 449.209,A -85,B 0,C 180,E1 -24522.399,E2 -24522.399} C_VEL
LIN {X 0,Y 363.591,Z 449.251,A -85,B 0,C 180,E1 -24524.537,E2 -24524.537} C_VEL
LIN {X 0,Y 364.38,Z 450.504,A -85,B 0,C 180,E1 -24526.615,E2 -24526.615} C_VEL
LIN {X 0,Y 364.584,Z 451.798,A -85,B 0,C 180,E1 -24527.27,E2 -24527.27} C_VEL
LIN {X 0,Y 364.298,Z 456.44,A -85,B 0,C 180,E1 -24528.077,E2 -24528.077} C_VEL
LIN {X 0,Y 361.734,Z 474.776,A -85,B 0,C 180,E1 -24529.676,E2 -24529.676} C_VEL
LIN {X 0,Y 359.544,Z 491.14,A -85,B 0,C 180,E1 -24530.917,E2 -24530.917} C_VEL
LIN {X 0,Y 358.067,Z 500.993,A -85,B 0,C 180,E1 -24531.47,E2 -24531.47} C_VEL
LIN {X 0,Y 352.657,Z 527.863,A -85,B 0,C 180,E1 -24532.445,E2 -24532.445} C_VEL
LIN {X 0,Y 347.685,Z 545.995,A -85,B 0,C 180,E1 -24533.267,E2 -24533.267} C_VEL
LIN {X 0,Y 342.297,Z 561.529,A -85,B 0,C 180,E1 -24534.143,E2 -24534.143} C_VEL
LIN {X 0,Y 336.878,Z 574.895,A -85,B 0,C 180,E1 -24535.125,E2 -24535.125} C_VEL
LIN {X 0,Y 330.599,Z 588.525,A -85,B 0,C 180,E1 -24536.391,E2 -24536.391} C_VEL
LIN {X 0,Y 324.652,Z 600.043,A -85,B 0,C 180,E1 -24537.724,E2 -24537.724} C_VEL
LIN {X 0,Y 317.706,Z 612.355,A -85,B 0,C 180,E1 -24539.53,E2 -24539.53} C_VEL
LIN {X 0,Y 312.315,Z 621.236,A -85,B 0,C 180,E1 -24541.171,E2 -24541.171} C_VEL
LIN {X 0,Y 305.912,Z 631.1,A -85,B 0,C 180,E1 -24543.481,E2 -24543.481} C_VEL
LIN {X 0,Y 300.439,Z 639.177,A -85,B 0,C 180,E1 -24545.921,E2 -24545.921} C_VEL
LIN {X 0,Y 295.703,Z 645.694,A -85,B 0,C 180,E1 -24548.459,E2 -24548.459} C_VEL
LIN {X 0,Y 291.984,Z 650.753,A -85,B 0,C 180,E1 -24551.104,E2 -24551.104} C_VEL
LIN {X 0,Y 289.92,Z 653.66,A -85,B 0,C 180,E1 -24553.147,E2 -24553.147} C_VEL
LIN {X 0,Y 288.022,Z 656.483,A -85,B 0,C 180,E1 -24555.925,E2 -24555.925} C_VEL
LIN {X 0,Y 287.098,Z 658.109,A -85,B 0,C 180,E1 -24558.566,E2 -24558.566} C_VEL
LIN {X 0,Y 286.992,Z 661.041,A -85,B 0,C 180,E1 -24560.473,E2 -24560.473} C_VEL
LIN {X 0,Y 286.542,Z 671.054,A -85,B 0,C 180,E1 -24562.626,E2 -24562.626} C_VEL
LIN {X 0,Y 286.414,Z 679.222,A -85,B 0,C 180,E1 -24564.738,E2 -24564.738} C_VEL
LIN {X 0,Y 286.236,Z 685.947,A -85,B 0,C 180,E1 -24566.843,E2 -24566.843} C_VEL
LIN {X 0,Y 286.112,Z 692.265,A -85,B 0,C 180,E1 -24569.298,E2 -24569.298} C_VEL
LIN {X 0,Y 285.893,Z 696.535,A -85,B 0,C 180,E1 -24571.404,E2 -24571.404} C_VEL
LIN {X 0,Y 285.858,Z 698.866,A -85,B 0,C 180,E1 -24572.809,E2 -24572.809} C_VEL
LIN {X 0,Y 285.956,Z 702.407,A -85,B 0,C 180,E1 -24575.623,E2 -24575.623} C_VEL
LIN {X 0,Y 286.557,Z 704.574,A -85,B 0,C 180,E1 -24578.433,E2 -24578.433} C_VEL
LIN {X 0,Y 287.97,Z 705.447,A -85,B 0,C 180,E1 -24581.22,E2 -24581.22} C_VEL
LIN {X 0,Y 290.139,Z 705.026,A -85,B 0,C 180,E1 -24583.97,E2 -24583.97} C_VEL
LIN {X 0,Y 293.241,Z 703.308,A -85,B 0,C 180,E1 -24586.656,E2 -24586.656} C_VEL
LIN {X 0,Y 296.748,Z 700.317,A -85,B 0,C 180,E1 -24589.296,E2 -24589.296} C_VEL
LIN {X 0,Y 301.225,Z 695.943,A -85,B 0,C 180,E1 -24591.842,E2 -24591.842} C_VEL
LIN {X 0,Y 306.496,Z 690.089,A -85,B 0,C 180,E1 -24594.29,E2 -24594.29} C_VEL
LIN {X 0,Y 312.371,Z 682.599,A -85,B 0,C 180,E1 -24596.645,E2 -24596.645} C_VEL
LIN {X 0,Y 318.159,Z 674.507,A -85,B 0,C 180,E1 -24598.609,E2 -24598.609} C_VEL
LIN {X 0,Y 323.434,Z 666.324,A -85,B 0,C 180,E1 -24600.233,E2 -24600.233} C_VEL
LIN {X 0,Y 330.123,Z 654.921,A -85,B 0,C 180,E1 -24602.035,E2 -24602.035} C_VEL
LIN {X 0,Y 336.037,Z 643.627,A -85,B 0,C 180,E1 -24603.458,E2 -24603.458} C_VEL
LIN {X 0,Y 341.672,Z 631.487,A -85,B 0,C 180,E1 -24604.673,E2 -24604.673} C_VEL
LIN {X 0,Y 346.898,Z 618.675,A -85,B 0,C 180,E1 -24605.699,E2 -24605.699} C_VEL
LIN {X 0,Y 351.589,Z 605.464,A -85,B 0,C 180,E1 -24606.525,E2 -24606.525} C_VEL
LIN {X 0,Y 355.661,Z 591.872,A -85,B 0,C 180,E1 -24607.183,E2 -24607.183} C_VEL
LIN {X 0,Y 359.62,Z 574.82,A -85,B 0,C 180,E1 -24607.846,E2 -24607.846} C_VEL
LIN {X 0,Y 374.797,Z 503.882,A -85,B 0,C 180,E1 -24610.359,E2 -24610.359} C_VEL
LIN {X 0,Y 377.256,Z 490.441,A -85,B 0,C 180,E1 -24611.322,E2 -24611.322} C_VEL
LIN {X 0,Y 377.583,Z 488.609,A -85,B 0,C 180,E1 -24611.483,E2 -24611.483} C_VEL
LIN {X 0,Y 377.192,Z 488.264,A -85,B 0,C 180,E1 -24612.03,E2 -24612.03} C_VEL
LIN {X 0,Y 376.124,Z 488.356,A -85,B 0,C 180,E1 -24614.128,E2 -24614.128} C_VEL
LIN {X 0,Y 375.774,Z 489.572,A -85,B 0,C 180,E1 -24615.549,E2 -24615.549} C_VEL
LIN {X 0,Y 375.697,Z 492.278,A -85,B 0,C 180,E1 -24617.219,E2 -24617.219} C_VEL
LIN {X 0,Y 375.692,Z 494.466,A -85,B 0,C 180,E1 -24618.032,E2 -24618.032} C_VEL
LIN {X 0,Y 373.651,Z 507.982,A -85,B 0,C 180,E1 -24619.49,E2 -24619.49} C_VEL
LIN {X 0,Y 372.883,Z 513.013,A -85,B 0,C 180,E1 -24619.942,E2 -24619.942} C_VEL
LIN {X 0,Y 357.45,Z 585.327,A -85,B 0,C 180,E1 -24622.506,E2 -24622.506} C_VEL
LIN {X 0,Y 353.373,Z 600.021,A -85,B 0,C 180,E1 -24623.159,E2 -24623.159} C_VEL
LIN {X 0,Y 348.586,Z 614.266,A -85,B 0,C 180,E1 -24624.003,E2 -24624.003} C_VEL
LIN {X 0,Y 343.743,Z 626.723,A -85,B 0,C 180,E1 -24624.944,E2 -24624.944} C_VEL
LIN {X 0,Y 337.46,Z 640.584,A -85,B 0,C 180,E1 -24626.273,E2 -24626.273} C_VEL
LIN {X 0,Y 331.254,Z 652.739,A -85,B 0,C 180,E1 -24627.766,E2 -24627.766} C_VEL
LIN {X 0,Y 325.554,Z 662.674,A -85,B 0,C 180,E1 -24629.27,E2 -24629.27} C_VEL
LIN {X 0,Y 319.26,Z 672.551,A -85,B 0,C 180,E1 -24631.14,E2 -24631.14} C_VEL
LIN {X 0,Y 313.498,Z 680.747,A -85,B 0,C 180,E1 -24633.1,E2 -24633.1} C_VEL
LIN {X 0,Y 308.181,Z 687.533,A -85,B 0,C 180,E1 -24635.136,E2 -24635.136} C_VEL
LIN {X 0,Y 302.864,Z 693.715,A -85,B 0,C 180,E1 -24637.567,E2 -24637.567} C_VEL
LIN {X 0,Y 299.229,Z 697.403,A -85,B 0,C 180,E1 -24639.444,E2 -24639.444} C_VEL
LIN {X 0,Y 295.199,Z 701.046,A -85,B 0,C 180,E1 -24642.034,E2 -24642.034} C_VEL
LIN {X 0,Y 291.843,Z 703.373,A -85,B 0,C 180,E1 -24644.692,E2 -24644.692} C_VEL
LIN {X 0,Y 289.173,Z 704.416,A -85,B 0,C 180,E1 -24647.409,E2 -24647.409} C_VEL
LIN {X 0,Y 287.287,Z 704.173,A -85,B 0,C 180,E1 -24650.174,E2 -24650.174} C_VEL
LIN {X 0,Y 286.273,Z 702.643,A -85,B 0,C 180,E1 -24652.973,E2 -24652.973} C_VEL
LIN {X 0,Y 285.745,Z 699.782,A -85,B 0,C 180,E1 -24655.783,E2 -24655.783} C_VEL
LIN {X 0,Y 285.808,Z 695.521,A -85,B 0,C 180,E1 -24658.596,E2 -24658.596} C_VEL
LIN {X 0,Y 285.949,Z 691.265,A -85,B 0,C 180,E1 -24660.702,E2 -24660.702} C_VEL
LIN {X 0,Y 286.143,Z 685.01,A -85,B 0,C 180,E1 -24663.158,E2 -24663.158} C_VEL
LIN {X 0,Y 286.319,Z 678.365,A -85,B 0,C 180,E1 -24665.264,E2 -24665.264} C_VEL
LIN {X 0,Y 286.556,Z 670.338,A -85,B 0,C 180,E1 -24667.373,E2 -24667.373} C_VEL
LIN {X 0,Y 287.032,Z 660.717,A -85,B 0,C 180,E1 -24669.481,E2 -24669.481} C_VEL
LIN {X 0,Y 287.662,Z 649.056,A -85,B 0,C 180,E1 -24671.589,E2 -24671.589} C_VEL
LIN {X 0,Y 288.378,Z 637.643,A -85,B 0,C 180,E1 -24673.296,E2 -24673.296} C_VEL
LIN {X 0,Y 289.209,Z 624.473,A -85,B 0,C 180,E1 -24674.912,E2 -24674.912} C_VEL
LIN {X 0,Y 290.089,Z 610.496,A -85,B 0,C 180,E1 -24676.302,E2 -24676.302} C_VEL
LIN {X 0,Y 290.791,Z 596.063,A -85,B 0,C 180,E1 -24677.433,E2 -24677.433} C_VEL
LIN {X 0,Y 291.557,Z 580.473,A -85,B 0,C 180,E1 -24678.335,E2 -24678.335} C_VEL
LIN {X 0,Y 295.257,Z 478.239,A -85,B 0,C 180,E1 -24682.56,E2 -24682.56} C_VEL
LIN {X 0,Y 293.102,Z 450.396,A -85,B 0,C 180,E1 -24683.737,E2 -24683.737} C_VEL
LIN {X 0,Y 292.863,Z 439.44,A -85,B 0,C 180,E1 -24684.227,E2 -24684.227} C_VEL
LIN {X 0,Y 295.625,Z 412.173,A -85,B 0,C 180,E1 -24688.757,E2 -24688.757} C_VEL
LIN {X 0,Y 296.844,Z 400.549,A -85,B 0,C 180,E1 -24690.682,E2 -24690.682} C_VEL
LIN {X 0,Y 293.896,Z 386.341,A -85,B 0,C 180,E1 -24693.242,E2 -24693.242} C_VEL
LIN {X 0,Y 289.396,Z 366.188,A -85,B 0,C 180,E1 -24696.992,E2 -24696.992} C_VEL
LIN {X 0,Y 288.527,Z 362.103,A -85,B 0,C 180,E1 -24697.806,E2 -24697.806} C_VEL
LIN {X 0,Y 288.436,Z 362.107,A -85,B 0,C 180,E1 -24701.166,E2 -24701.166} C_VEL
LIN {X 0,Y 288.473,Z 362.102,A -85,B 0,C 180,E1 -24705.239,E2 -24705.239} C_VEL
LIN {X 0,Y 288.444,Z 362.107,A -85,B 0,C 180,E1 -24709.031,E2 -24709.031} C_VEL
LIN {X 0,Y 288.458,Z 362.104,A -85,B 0,C 180,E1 -24713.257,E2 -24713.257} C_VEL
LIN {X 0,Y 288.451,Z 362.11,A -85,B 0,C 180,E1 -24716.047,E2 -24716.047} C_VEL
LIN {X 0,Y 288.458,Z 362.095,A -85,B 0,C 180,E1 -24719.341,E2 -24719.341} C_VEL
LIN {X 0,Y 288.491,Z 362.186,A -85,B 0,C 180,E1 -24723.548,E2 -24723.548} C_VEL
LIN {X 0,Y 289.484,Z 364.933,A -85,B 0,C 180,E1 -24723.739,E2 -24723.739} C_VEL
LIN {X 0,Y 296.353,Z 377.848,A -85,B 0,C 180,E1 -24724.848,E2 -24724.848} C_VEL
LIN {X 0,Y 304.914,Z 396.356,A -85,B 0,C 180,E1 -24726.209,E2 -24726.209} C_VEL
LIN {X 0,Y 307.377,Z 402.624,A -85,B 0,C 180,E1 -24726.608,E2 -24726.608} C_VEL
LIN {X 0,Y 305.506,Z 464.275,A -85,B 0,C 180,E1 -24728.015,E2 -24728.015} C_VEL
LIN {X 0,Y 305.15,Z 482.905,A -85,B 0,C 180,E1 -24728.541,E2 -24728.541} C_VEL
LIN {X 0,Y 304.497,Z 496.989,A -85,B 0,C 180,E1 -24729.2,E2 -24729.2} C_VEL
LIN {X 0,Y 303.41,Z 510.585,A -85,B 0,C 180,E1 -24730.092,E2 -24730.092} C_VEL
LIN {X 0,Y 301.913,Z 523.703,A -85,B 0,C 180,E1 -24731.222,E2 -24731.222} C_VEL
LIN {X 0,Y 300.455,Z 535.535,A -85,B 0,C 180,E1 -24732.533,E2 -24732.533} C_VEL
LIN {X 0,Y 298.698,Z 546.678,A -85,B 0,C 180,E1 -24734.041,E2 -24734.041} C_VEL
LIN {X 0,Y 296.877,Z 556.599,A -85,B 0,C 180,E1 -24735.666,E2 -24735.666} C_VEL
LIN {X 0,Y 294.809,Z 566.61,A -85,B 0,C 180,E1 -24737.653,E2 -24737.653} C_VEL
LIN {X 0,Y 293.076,Z 574.932,A -85,B 0,C 180,E1 -24739.674,E2 -24739.674} C_VEL
LIN {X 0,Y 291.38,Z 582.884,A -85,B 0,C 180,E1 -24742.055,E2 -24742.055} C_VEL
LIN {X 0,Y 289.99,Z 589.309,A -85,B 0,C 180,E1 -24744.456,E2 -24744.456} C_VEL
LIN {X 0,Y 288.899,Z 595.009,A -85,B 0,C 180,E1 -24747.221,E2 -24747.221} C_VEL
LIN {X 0,Y 288.122,Z 599.196,A -85,B 0,C 180,E1 -24750,E2 -24750} C_VEL
LIN {X 0,Y 287.785,Z 601.983,A -85,B 0,C 180,E1 -24752.79,E2 -24752.79} C_VEL
LIN {X 0,Y 287.882,Z 603.446,A -85,B 0,C 180,E1 -24755.585,E2 -24755.585} C_VEL
LIN {X 0,Y 288.25,Z 603.63,A -85,B 0,C 180,E1 -24758.384,E2 -24758.384} C_VEL
LIN {X 0,Y 288.995,Z 602.524,A -85,B 0,C 180,E1 -24761.181,E2 -24761.181} C_VEL
LIN {X 0,Y 290.275,Z 600.073,A -85,B 0,C 180,E1 -24763.964,E2 -24763.964} C_VEL
LIN {X 0,Y 292.012,Z 596.19,A -85,B 0,C 180,E1 -24766.729,E2 -24766.729} C_VEL
LIN {X 0,Y 294.173,Z 590.765,A -85,B 0,C 180,E1 -24769.472,E2 -24769.472} C_VEL
LIN {X 0,Y 296.115,Z 585.598,A -85,B 0,C 180,E1 -24771.509,E2 -24771.509} C_VEL
LIN {X 0,Y 298.711,Z 578.111,A -85,B 0,C 180,E1 -24773.863,E2 -24773.863} C_VEL
LIN {X 0,Y 301.266,Z 570.292,A -85,B 0,C 180,E1 -24775.845,E2 -24775.845} C_VEL
LIN {X 0,Y 304.11,Z 560.811,A -85,B 0,C 180,E1 -24777.802,E2 -24777.802} C_VEL
LIN {X 0,Y 306.646,Z 550.772,A -85,B 0,C 180,E1 -24779.513,E2 -24779.513} C_VEL
LIN {X 0,Y 309.15,Z 539.841,A -85,B 0,C 180,E1 -24781.028,E2 -24781.028} C_VEL
LIN {X 0,Y 311.743,Z 527.031,A -85,B 0,C 180,E1 -24782.442,E2 -24782.442} C_VEL
LIN {X 0,Y 313.67,Z 513.442,A -85,B 0,C 180,E1 -24783.648,E2 -24783.648} C_VEL
LIN {X 0,Y 315.13,Z 500.196,A -85,B 0,C 180,E1 -24784.533,E2 -24784.533} C_VEL
LIN {X 0,Y 316.166,Z 486.294,A -85,B 0,C 180,E1 -24785.201,E2 -24785.201} C_VEL
LIN {X 0,Y 316.642,Z 470.984,A -85,B 0,C 180,E1 -24785.675,E2 -24785.675} C_VEL
LIN {X 0,Y 318.711,Z 415.755,A -85,B 0,C 180,E1 -24786.901,E2 -24786.901} C_VEL
LIN {X 0,Y 310.158,Z 398.878,A -85,B 0,C 180,E1 -24788.484,E2 -24788.484} C_VEL
LIN {X 0,Y 302.119,Z 384.613,A -85,B 0,C 180,E1 -24790.039,E2 -24790.039} C_VEL
LIN {X 0,Y 292.948,Z 370.036,A -85,B 0,C 180,E1 -24791.91,E2 -24791.91} C_VEL
LIN {X 0,Y 290.552,Z 366.333,A -85,B 0,C 180,E1 -24792.424,E2 -24792.424} C_VEL
LIN {X 0,Y 288.963,Z 364.139,A -85,B 0,C 180,E1 -24792.764,E2 -24792.764} C_VEL
LIN {X 0,Y 288.413,Z 362.119,A -85,B 0,C 180,E1 -24792.964,E2 -24792.964} C_VEL
LIN {X 0,Y 288.397,Z 362.12,A -85,B 0,C 180,E1 -24796.772,E2 -24796.772} C_VEL
LIN {X 0,Y 288.388,Z 362.101,A -85,B 0,C 180,E1 -24800.839,E2 -24800.839} C_VEL
LIN {X 0,Y 288.416,Z 362.069,A -85,B 0,C 180,E1 -24804.347,E2 -24804.347} C_VEL
LIN {X 0,Y 288.429,Z 362.106,A -85,B 0,C 180,E1 -24808.209,E2 -24808.209} C_VEL
LIN {X 0,Y 288.472,Z 362.105,A -85,B 0,C 180,E1 -24812.526,E2 -24812.526} C_VEL
LIN {X 0,Y 288.578,Z 362.228,A -85,B 0,C 180,E1 -24816.329,E2 -24816.329} C_VEL
LIN {X 0,Y 293.58,Z 382.885,A -85,B 0,C 180,E1 -24817.265,E2 -24817.265} C_VEL
LIN {X 0,Y 294.479,Z 386.915,A -85,B 0,C 180,E1 -24817.443,E2 -24817.443} C_VEL
LIN {X 0,Y 292.018,Z 467.62,A -85,B 0,C 180,E1 -24820.651,E2 -24820.651} C_VEL
LIN {X 0,Y 291.588,Z 484.708,A -85,B 0,C 180,E1 -24821.44,E2 -24821.44} C_VEL
LIN {X 0,Y 290.936,Z 500.707,A -85,B 0,C 180,E1 -24822.485,E2 -24822.485} C_VEL
LIN {X 0,Y 290.69,Z 506.052,A -85,B 0,C 180,E1 -24822.908,E2 -24822.908} C_VEL
LIN {X 0,Y 289.745,Z 511.405,A -85,B 0,C 180,E1 -24823.368,E2 -24823.368} C_VEL
LIN {X 0,Y 286.388,Z 519.789,A -85,B 0,C 180,E1 -24824.189,E2 -24824.189} C_VEL
LIN {X 0,Y 283.067,Z 527.938,A -85,B 0,C 180,E1 -24825.121,E2 -24825.121} C_VEL
LIN {X 0,Y 282.185,Z 532.924,A -85,B 0,C 180,E1 -24825.744,E2 -24825.744} C_VEL
LIN {X 0,Y 281.48,Z 546.095,A -85,B 0,C 180,E1 -24827.606,E2 -24827.606} C_VEL
LIN {X 0,Y 280.793,Z 557.656,A -85,B 0,C 180,E1 -24829.58,E2 -24829.58} C_VEL
LIN {X 0,Y 280.295,Z 568.243,A -85,B 0,C 180,E1 -24831.738,E2 -24831.738} C_VEL
LIN {X 0,Y 279.961,Z 578.419,A -85,B 0,C 180,E1 -24834.256,E2 -24834.256} C_VEL
LIN {X 0,Y 279.968,Z 586.784,A -85,B 0,C 180,E1 -24836.773,E2 -24836.773} C_VEL
LIN {X 0,Y 280.193,Z 594.034,A -85,B 0,C 180,E1 -24839.445,E2 -24839.445} C_VEL
LIN {X 0,Y 280.876,Z 599.801,A -85,B 0,C 180,E1 -24842.143,E2 -24842.143} C_VEL
LIN {X 0,Y 281.802,Z 603.421,A -85,B 0,C 180,E1 -24844.276,E2 -24844.276} C_VEL
LIN {X 0,Y 283.528,Z 606.985,A -85,B 0,C 180,E1 -24847.095,E2 -24847.095} C_VEL
LIN {X 0,Y 285.792,Z 609.164,A -85,B 0,C 180,E1 -24849.878,E2 -24849.878} C_VEL
LIN {X 0,Y 288.721,Z 610.001,A -85,B 0,C 180,E1 -24852.611,E2 -24852.611} C_VEL
LIN {X 0,Y 292.697,Z 609.429,A -85,B 0,C 180,E1 -24855.262,E2 -24855.262} C_VEL
LIN {X 0,Y 297.078,Z 607.522,A -85,B 0,C 180,E1 -24857.849,E2 -24857.849} C_VEL
LIN {X 0,Y 301.923,Z 604.281,A -85,B 0,C 180,E1 -24860.364,E2 -24860.364} C_VEL
LIN {X 0,Y 305.954,Z 600.841,A -85,B 0,C 180,E1 -24862.194,E2 -24862.194} C_VEL
LIN {X 0,Y 311.828,Z 594.898,A -85,B 0,C 180,E1 -24864.554,E2 -24864.554} C_VEL
LIN {X 0,Y 317.299,Z 588.322,A -85,B 0,C 180,E1 -24866.553,E2 -24866.553} C_VEL
LIN {X 0,Y 323.187,Z 580.154,A -85,B 0,C 180,E1 -24868.477,E2 -24868.477} C_VEL
LIN {X 0,Y 329.464,Z 570.19,A -85,B 0,C 180,E1 -24870.326,E2 -24870.326} C_VEL
LIN {X 0,Y 336.056,Z 557.976,A -85,B 0,C 180,E1 -24872.106,E2 -24872.106} C_VEL
LIN {X 0,Y 341.452,Z 546.307,A -85,B 0,C 180,E1 -24873.456,E2 -24873.456} C_VEL
LIN {X 0,Y 346.835,Z 532.302,A -85,B 0,C 180,E1 -24874.786,E2 -24874.786} C_VEL
LIN {X 0,Y 351.364,Z 518.094,A -85,B 0,C 180,E1 -24875.845,E2 -24875.845} C_VEL
LIN {X 0,Y 354.819,Z 504.079,A -85,B 0,C 180,E1 -24876.667,E2 -24876.667} C_VEL
LIN {X 0,Y 359.674,Z 480.153,A -85,B 0,C 180,E1 -24877.699,E2 -24877.699} C_VEL
LIN {X 0,Y 363.767,Z 460.466,A -85,B 0,C 180,E1 -24878.422,E2 -24878.422} C_VEL
LIN {X 0,Y 362.588,Z 457.063,A -85,B 0,C 180,E1 -24880.4,E2 -24880.4} C_VEL
LIN {X 0,Y 361.803,Z 456.028,A -85,B 0,C 180,E1 -24882.656,E2 -24882.656} C_VEL
LIN {X 0,Y 361.87,Z 456.185,A -85,B 0,C 180,E1 -24884.661,E2 -24884.661} C_VEL
LIN {X 0,Y 362.515,Z 457.301,A -85,B 0,C 180,E1 -24886.442,E2 -24886.442} C_VEL
LIN {X 0,Y 362.566,Z 458.063,A -85,B 0,C 180,E1 -24886.758,E2 -24886.758} C_VEL
LIN {X 0,Y 362.233,Z 460.899,A -85,B 0,C 180,E1 -24887.236,E2 -24887.236} C_VEL
LIN {X 0,Y 359.256,Z 479.731,A -85,B 0,C 180,E1 -24888.882,E2 -24888.882} C_VEL
LIN {X 0,Y 356.923,Z 495.261,A -85,B 0,C 180,E1 -24890.017,E2 -24890.017} C_VEL
LIN {X 0,Y 355.498,Z 503.547,A -85,B 0,C 180,E1 -24890.464,E2 -24890.464} C_VEL
LIN {X 0,Y 350.015,Z 528.743,A -85,B 0,C 180,E1 -24891.382,E2 -24891.382} C_VEL
LIN {X 0,Y 345.331,Z 544.902,A -85,B 0,C 180,E1 -24892.115,E2 -24892.115} C_VEL
LIN {X 0,Y 339.951,Z 559.688,A -85,B 0,C 180,E1 -24892.938,E2 -24892.938} C_VEL
LIN {X 0,Y 333.677,Z 574.489,A -85,B 0,C 180,E1 -24894.001,E2 -24894.001} C_VEL
LIN {X 0,Y 327.151,Z 587.91,A -85,B 0,C 180,E1 -24895.246,E2 -24895.246} C_VEL
LIN {X 0,Y 320.983,Z 599.237,A -85,B 0,C 180,E1 -24896.564,E2 -24896.564} C_VEL
LIN {X 0,Y 314.715,Z 609.83,A -85,B 0,C 180,E1 -24898.089,E2 -24898.089} C_VEL
LIN {X 0,Y 308.009,Z 620.201,A -85,B 0,C 180,E1 -24899.98,E2 -24899.98} C_VEL
LIN {X 0,Y 302.016,Z 628.915,A -85,B 0,C 180,E1 -24901.988,E2 -24901.988} C_VEL
LIN {X 0,Y 296.693,Z 636.186,A -85,B 0,C 180,E1 -24904.103,E2 -24904.103} C_VEL
LIN {X 0,Y 291.492,Z 643.011,A -85,B 0,C 180,E1 -24906.641,E2 -24906.641} C_VEL
LIN {X 0,Y 287.07,Z 648.382,A -85,B 0,C 180,E1 -24909.28,E2 -24909.28} C_VEL
LIN {X 0,Y 284.442,Z 651.576,A -85,B 0,C 180,E1 -24911.329,E2 -24911.329} C_VEL
LIN {X 0,Y 281.973,Z 654.701,A -85,B 0,C 180,E1 -24914.142,E2 -24914.142} C_VEL
LIN {X 0,Y 280.372,Z 656.611,A -85,B 0,C 180,E1 -24917.006,E2 -24917.006} C_VEL
LIN {X 0,Y 280.083,Z 657.179,A -85,B 0,C 180,E1 -24918.126,E2 -24918.126} C_VEL
LIN {X 0,Y 279.936,Z 661.08,A -85,B 0,C 180,E1 -24920.776,E2 -24920.776} C_VEL
LIN {X 0,Y 279.536,Z 670.333,A -85,B 0,C 180,E1 -24922.802,E2 -24922.802} C_VEL
LIN {X 0,Y 279.405,Z 678.572,A -85,B 0,C 180,E1 -24924.966,E2 -24924.966} C_VEL
LIN {X 0,Y 279.22,Z 685.359,A -85,B 0,C 180,E1 -24927.124,E2 -24927.124} C_VEL
LIN {X 0,Y 279.12,Z 690.968,A -85,B 0,C 180,E1 -24929.281,E2 -24929.281} C_VEL
LIN {X 0,Y 278.877,Z 695.465,A -85,B 0,C 180,E1 -24931.439,E2 -24931.439} C_VEL
LIN {X 0,Y 278.814,Z 699.014,A -85,B 0,C 180,E1 -24933.601,E2 -24933.601} C_VEL
LIN {X 0,Y 278.931,Z 701.76,A -85,B 0,C 180,E1 -24935.765,E2 -24935.765} C_VEL
LIN {X 0,Y 279.531,Z 704.198,A -85,B 0,C 180,E1 -24938.647,E2 -24938.647} C_VEL
LIN {X 0,Y 281.018,Z 705.355,A -85,B 0,C 180,E1 -24941.502,E2 -24941.502} C_VEL
LIN {X 0,Y 283.264,Z 705.235,A -85,B 0,C 180,E1 -24944.316,E2 -24944.316} C_VEL
LIN {X 0,Y 286.474,Z 703.834,A -85,B 0,C 180,E1 -24947.062,E2 -24947.062} C_VEL
LIN {X 0,Y 290.113,Z 701.178,A -85,B 0,C 180,E1 -24949.756,E2 -24949.756} C_VEL
LIN {X 0,Y 294.747,Z 697.162,A -85,B 0,C 180,E1 -24952.348,E2 -24952.348} C_VEL
LIN {X 0,Y 300.191,Z 691.701,A -85,B 0,C 180,E1 -24954.834,E2 -24954.834} C_VEL
LIN {X 0,Y 306.275,Z 684.712,A -85,B 0,C 180,E1 -24957.219,E2 -24957.219} C_VEL
LIN {X 0,Y 312.229,Z 677.149,A -85,B 0,C 180,E1 -24959.205,E2 -24959.205} C_VEL
LIN {X 0,Y 318.627,Z 668.078,A -85,B 0,C 180,E1 -24961.105,E2 -24961.105} C_VEL
LIN {X 0,Y 325.547,Z 657.086,A -85,B 0,C 180,E1 -24962.907,E2 -24962.907} C_VEL
LIN {X 0,Y 331.722,Z 646.098,A -85,B 0,C 180,E1 -24964.344,E2 -24964.344} C_VEL
LIN {X 0,Y 338.053,Z 633.495,A -85,B 0,C 180,E1 -24965.644,E2 -24965.644} C_VEL
LIN {X 0,Y 343.321,Z 621.532,A -85,B 0,C 180,E1 -24966.638,E2 -24966.638} C_VEL
LIN {X 0,Y 348.889,Z 606.818,A -85,B 0,C 180,E1 -24967.577,E2 -24967.577} C_VEL
LIN {X 0,Y 353.406,Z 592.545,A -85,B 0,C 180,E1 -24968.27,E2 -24968.27} C_VEL
LIN {X 0,Y 357.52,Z 575.911,A -85,B 0,C 180,E1 -24968.915,E2 -24968.915} C_VEL
LIN {X 0,Y 373.2,Z 505.741,A -85,B 0,C 180,E1 -24971.382,E2 -24971.382} C_VEL
LIN {X 0,Y 375.312,Z 495.188,A -85,B 0,C 180,E1 -24972.134,E2 -24972.134} C_VEL
LIN {X 0,Y 374.347,Z 495.223,A -85,B 0,C 180,E1 -24974.085,E2 -24974.085} C_VEL
LIN {X 0,Y 373.921,Z 496.785,A -85,B 0,C 180,E1 -24975.688,E2 -24975.688} C_VEL
LIN {X 0,Y 373.802,Z 498.949,A -85,B 0,C 180,E1 -24976.953,E2 -24976.953} C_VEL
LIN {X 0,Y 373.745,Z 500.148,A -85,B 0,C 180,E1 -24977.368,E2 -24977.368} C_VEL
LIN {X 0,Y 371.686,Z 511.848,A -85,B 0,C 180,E1 -24978.621,E2 -24978.621} C_VEL
LIN {X 0,Y 371.014,Z 515.601,A -85,B 0,C 180,E1 -24978.947,E2 -24978.947} C_VEL
LIN {X 0,Y 355.567,Z 584.885,A -85,B 0,C 180,E1 -24981.375,E2 -24981.375} C_VEL
LIN {X 0,Y 350.731,Z 601.509,A -85,B 0,C 180,E1 -24982.113,E2 -24982.113} C_VEL
LIN {X 0,Y 345.182,Z 616.925,A -85,B 0,C 180,E1 -24983.048,E2 -24983.048} C_VEL
LIN {X 0,Y 340.454,Z 628.226,A -85,B 0,C 180,E1 -24983.919,E2 -24983.919} C_VEL
LIN {X 0,Y 334.102,Z 641.493,A -85,B 0,C 180,E1 -24985.207,E2 -24985.207} C_VEL
LIN {X 0,Y 327.855,Z 653.036,A -85,B 0,C 180,E1 -24986.624,E2 -24986.624} C_VEL
LIN {X 0,Y 321.823,Z 663.001,A -85,B 0,C 180,E1 -24988.143,E2 -24988.143} C_VEL
LIN {X 0,Y 315.167,Z 672.792,A -85,B 0,C 180,E1 -24989.997,E2 -24989.997} C_VEL
LIN {X 0,Y 309.067,Z 680.92,A -85,B 0,C 180,E1 -24991.949,E2 -24991.949} C_VEL
LIN {X 0,Y 303.45,Z 687.642,A -85,B 0,C 180,E1 -24993.988,E2 -24993.988} C_VEL
LIN {X 0,Y 297.759,Z 693.78,A -85,B 0,C 180,E1 -24996.428,E2 -24996.428} C_VEL
LIN {X 0,Y 292.681,Z 698.47,A -85,B 0,C 180,E1 -24998.963,E2 -24998.963} C_VEL
LIN {X 0,Y 288.488,Z 701.764,A -85,B 0,C 180,E1 -25001.601,E2 -25001.601} C_VEL
LIN {X 0,Y 285.015,Z 703.771,A -85,B 0,C 180,E1 -25004.316,E2 -25004.316} C_VEL
LIN {X 0,Y 282.237,Z 704.509,A -85,B 0,C 180,E1 -25007.094,E2 -25007.094} C_VEL
LIN {X 0,Y 280.302,Z 703.971,A -85,B 0,C 180,E1 -25009.926,E2 -25009.926} C_VEL
LIN {X 0,Y 279.232,Z 702.167,A -85,B 0,C 180,E1 -25012.795,E2 -25012.795} C_VEL
LIN {X 0,Y 278.706,Z 699.042,A -85,B 0,C 180,E1 -25015.676,E2 -25015.676} C_VEL
LIN {X 0,Y 278.8,Z 694.494,A -85,B 0,C 180,E1 -25018.561,E2 -25018.561} C_VEL
LIN {X 0,Y 278.963,Z 690.002,A -85,B 0,C 180,E1 -25020.72,E2 -25020.72} C_VEL
LIN {X 0,Y 279.162,Z 683.445,A -85,B 0,C 180,E1 -25023.237,E2 -25023.237} C_VEL
LIN {X 0,Y 279.385,Z 675.24,A -85,B 0,C 180,E1 -25025.756,E2 -25025.756} C_VEL
LIN {X 0,Y 279.662,Z 666.611,A -85,B 0,C 180,E1 -25027.918,E2 -25027.918} C_VEL
LIN {X 0,Y 280.202,Z 656.214,A -85,B 0,C 180,E1 -25030.078,E2 -25030.078} C_VEL
LIN {X 0,Y 280.961,Z 643.626,A -85,B 0,C 180,E1 -25032.235,E2 -25032.235} C_VEL
LIN {X 0,Y 281.7,Z 630.562,A -85,B 0,C 180,E1 -25034.051,E2 -25034.051} C_VEL
LIN {X 0,Y 282.631,Z 616.477,A -85,B 0,C 180,E1 -25035.636,E2 -25035.636} C_VEL
LIN {X 0,Y 283.423,Z 602.589,A -85,B 0,C 180,E1 -25036.882,E2 -25036.882} C_VEL
LIN {X 0,Y 284.16,Z 586.18,A -85,B 0,C 180,E1 -25037.993,E2 -25037.993} C_VEL
LIN {X 0,Y 284.956,Z 566.902,A -85,B 0,C 180,E1 -25038.915,E2 -25038.915} C_VEL
LIN {X 0,Y 288.147,Z 478.316,A -85,B 0,C 180,E1 -25042.67,E2 -25042.67} C_VEL
LIN {X 0,Y 285.997,Z 448.922,A -85,B 0,C 180,E1 -25043.956,E2 -25043.956} C_VEL
LIN {X 0,Y 285.813,Z 439.524,A -85,B 0,C 180,E1 -25044.381,E2 -25044.381} C_VEL
LIN {X 0,Y 288.548,Z 413.122,A -85,B 0,C 180,E1 -25048.847,E2 -25048.847} C_VEL
LIN {X 0,Y 289.787,Z 400.964,A -85,B 0,C 180,E1 -25050.901,E2 -25050.901} C_VEL
LIN {X 0,Y 285.478,Z 381.071,A -85,B 0,C 180,E1 -25054.58,E2 -25054.58} C_VEL
LIN {X 0,Y 281.474,Z 362.981,A -85,B 0,C 180,E1 -25058.055,E2 -25058.055} C_VEL
LIN {X 0,Y 281.373,Z 362.99,A -85,B 0,C 180,E1 -25062.232,E2 -25062.232} C_VEL
LIN {X 0,Y 281.408,Z 362.983,A -85,B 0,C 180,E1 -25066.207,E2 -25066.207} C_VEL
LIN {X 0,Y 281.366,Z 362.988,A -85,B 0,C 180,E1 -25070.51,E2 -25070.51} C_VEL
LIN {X 0,Y 281.408,Z 362.981,A -85,B 0,C 180,E1 -25073.318,E2 -25073.318} C_VEL
LIN {X 0,Y 281.371,Z 362.982,A -85,B 0,C 180,E1 -25076.793,E2 -25076.793} C_VEL
LIN {X 0,Y 281.398,Z 362.989,A -85,B 0,C 180,E1 -25080.6,E2 -25080.6} C_VEL
LIN {X 0,Y 281.436,Z 362.989,A -85,B 0,C 180,E1 -25082.739,E2 -25082.739} C_VEL
LIN {X 0,Y 282.438,Z 365.835,A -85,B 0,C 180,E1 -25082.942,E2 -25082.942} C_VEL
LIN {X 0,Y 289.499,Z 378.852,A -85,B 0,C 180,E1 -25084.13,E2 -25084.13} C_VEL
LIN {X 0,Y 298.273,Z 397.496,A -85,B 0,C 180,E1 -25085.577,E2 -25085.577} C_VEL
LIN {X 0,Y 300.868,Z 403.777,A -85,B 0,C 180,E1 -25086.005,E2 -25086.005} C_VEL
LIN {X 0,Y 299.097,Z 468.21,A -85,B 0,C 180,E1 -25087.529,E2 -25087.529} C_VEL
LIN {X 0,Y 298.719,Z 484.319,A -85,B 0,C 180,E1 -25088.01,E2 -25088.01} C_VEL
LIN {X 0,Y 298.034,Z 498.185,A -85,B 0,C 180,E1 -25088.682,E2 -25088.682} C_VEL
LIN {X 0,Y 296.803,Z 512.234,A -85,B 0,C 180,E1 -25089.629,E2 -25089.629} C_VEL
LIN {X 0,Y 295.282,Z 525.122,A -85,B 0,C 180,E1 -25090.784,E2 -25090.784} C_VEL
LIN {X 0,Y 293.581,Z 538.089,A -85,B 0,C 180,E1 -25092.29,E2 -25092.29} C_VEL
LIN {X 0,Y 291.646,Z 549.751,A -85,B 0,C 180,E1 -25093.966,E2 -25093.966} C_VEL
LIN {X 0,Y 289.677,Z 559.572,A -85,B 0,C 180,E1 -25095.675,E2 -25095.675} C_VEL
LIN {X 0,Y 287.653,Z 569.118,A -85,B 0,C 180,E1 -25097.698,E2 -25097.698} C_VEL
LIN {X 0,Y 285.934,Z 577.14,A -85,B 0,C 180,E1 -25099.77,E2 -25099.77} C_VEL
LIN {X 0,Y 284.161,Z 584.838,A -85,B 0,C 180,E1 -25102.208,E2 -25102.208} C_VEL
LIN {X 0,Y 282.991,Z 590.23,A -85,B 0,C 180,E1 -25104.318,E2 -25104.318} C_VEL
LIN {X 0,Y 281.877,Z 595.893,A -85,B 0,C 180,E1 -25107.152,E2 -25107.152} C_VEL
LIN {X 0,Y 281.055,Z 600.051,A -85,B 0,C 180,E1 -25110,E2 -25110} C_VEL
LIN {X 0,Y 280.729,Z 602.805,A -85,B 0,C 180,E1 -25112.861,E2 -25112.861} C_VEL
LIN {X 0,Y 280.844,Z 604.238,A -85,B 0,C 180,E1 -25115.726,E2 -25115.726} C_VEL
LIN {X 0,Y 281.255,Z 604.391,A -85,B 0,C 180,E1 -25118.594,E2 -25118.594} C_VEL
LIN {X 0,Y 282.043,Z 603.252,A -85,B 0,C 180,E1 -25121.46,E2 -25121.46} C_VEL
LIN {X 0,Y 283.387,Z 600.76,A -85,B 0,C 180,E1 -25124.31,E2 -25124.31} C_VEL
LIN {X 0,Y 285.195,Z 596.841,A -85,B 0,C 180,E1 -25127.141,E2 -25127.141} C_VEL
LIN {X 0,Y 287.477,Z 591.379,A -85,B 0,C 180,E1 -25129.945,E2 -25129.945} C_VEL
LIN {X 0,Y 289.505,Z 586.172,A -85,B 0,C 180,E1 -25132.026,E2 -25132.026} C_VEL
LIN {X 0,Y 292.094,Z 579.019,A -85,B 0,C 180,E1 -25134.321,E2 -25134.321} C_VEL
LIN {X 0,Y 294.877,Z 570.772,A -85,B 0,C 180,E1 -25136.448,E2 -25136.448} C_VEL
LIN {X 0,Y 297.831,Z 561.233,A -85,B 0,C 180,E1 -25138.441,E2 -25138.441} C_VEL
LIN {X 0,Y 300.618,Z 550.382,A -85,B 0,C 180,E1 -25140.3,E2 -25140.3} C_VEL
LIN {X 0,Y 303.378,Z 538.819,A -85,B 0,C 180,E1 -25141.88,E2 -25141.88} C_VEL
LIN {X 0,Y 305.76,Z 527.177,A -85,B 0,C 180,E1 -25143.157,E2 -25143.157} C_VEL
LIN {X 0,Y 307.611,Z 514.42,A -85,B 0,C 180,E1 -25144.303,E2 -25144.303} C_VEL
LIN {X 0,Y 309.211,Z 500.309,A -85,B 0,C 180,E1 -25145.258,E2 -25145.258} C_VEL
LIN {X 0,Y 310.272,Z 485.944,A -85,B 0,C 180,E1 -25145.942,E2 -25145.942} C_VEL
LIN {X 0,Y 310.848,Z 469.215,A -85,B 0,C 180,E1 -25146.437,E2 -25146.437} C_VEL
LIN {X 0,Y 312.823,Z 418.026,A -85,B 0,C 180,E1 -25147.593,E2 -25147.593} C_VEL
LIN {X 0,Y 303.807,Z 400.273,A -85,B 0,C 180,E1 -25149.333,E2 -25149.333} C_VEL
LIN {X 0,Y 295.361,Z 385.574,A -85,B 0,C 180,E1 -25151.042,E2 -25151.042} C_VEL
LIN {X 0,Y 286.336,Z 371.435,A -85,B 0,C 180,E1 -25152.981,E2 -25152.981} C_VEL
LIN {X 0,Y 283.559,Z 367.294,A -85,B 0,C 180,E1 -25153.607,E2 -25153.607} C_VEL
LIN {X 0,Y 281.854,Z 364.873,A -85,B 0,C 180,E1 -25153.997,E2 -25153.997} C_VEL
LIN {X 0,Y 281.354,Z 362.995,A -85,B 0,C 180,E1 -25154.193,E2 -25154.193} C_VEL
LIN {X 0,Y 281.329,Z 362.992,A -85,B 0,C 180,E1 -25158.326,E2 -25158.326} C_VEL
LIN {X 0,Y 281.369,Z 362.942,A -85,B 0,C 180,E1 -25162.809,E2 -25162.809} C_VEL
LIN {X 0,Y 281.36,Z 362.991,A -85,B 0,C 180,E1 -25166.791,E2 -25166.791} C_VEL
LIN {X 0,Y 281.38,Z 362.983,A -85,B 0,C 180,E1 -25170.606,E2 -25170.606} C_VEL
LIN {X 0,Y 281.445,Z 362.972,A -85,B 0,C 180,E1 -25174.97,E2 -25174.97} C_VEL
LIN {X 0,Y 281.536,Z 363.168,A -85,B 0,C 180,E1 -25176.219,E2 -25176.219} C_VEL
LIN {X 0,Y 286.74,Z 384.709,A -85,B 0,C 180,E1 -25177.219,E2 -25177.219} C_VEL
LIN {X 0,Y 287.398,Z 387.18,A -85,B 0,C 180,E1 -25177.332,E2 -25177.332} C_VEL
LIN {X 0,Y 284.925,Z 467.149,A -85,B 0,C 180,E1 -25180.617,E2 -25180.617} C_VEL
LIN {X 0,Y 284.494,Z 484.456,A -85,B 0,C 180,E1 -25181.425,E2 -25181.425} C_VEL
LIN {X 0,Y 283.845,Z 500.594,A -85,B 0,C 180,E1 -25182.497,E2 -25182.497} C_VEL
LIN {X 0,Y 283.231,Z 514.165,A -85,B 0,C 180,E1 -25183.661,E2 -25183.661} C_VEL
LIN {X 0,Y 282.404,Z 528.304,A -85,B 0,C 180,E1 -25185.176,E2 -25185.176} C_VEL
LIN {X 0,Y 282.185,Z 532.924,A -85,B 0,C 180,E1 -25185.744,E2 -25185.744} C_VEL
LIN {X 0,Y 281.315,Z 537.811,A -85,B 0,C 180,E1 -25186.395,E2 -25186.395} C_VEL
LIN {X 0,Y 278.049,Z 545.347,A -85,B 0,C 180,E1 -25187.53,E2 -25187.53} C_VEL
LIN {X 0,Y 274.706,Z 552.572,A -85,B 0,C 180,E1 -25188.776,E2 -25188.776} C_VEL
LIN {X 0,Y 273.731,Z 556.96,A -85,B 0,C 180,E1 -25189.589,E2 -25189.589} C_VEL
LIN {X 0,Y 273.193,Z 568.169,A -85,B 0,C 180,E1 -25191.893,E2 -25191.893} C_VEL
LIN {X 0,Y 272.906,Z 578.523,A -85,B 0,C 180,E1 -25194.476,E2 -25194.476} C_VEL
LIN {X 0,Y 272.918,Z 587.025,A -85,B 0,C 180,E1 -25197.057,E2 -25197.057} C_VEL
LIN {X 0,Y 273.086,Z 593.062,A -85,B 0,C 180,E1 -25199.265,E2 -25199.265} C_VEL
LIN {X 0,Y 273.779,Z 599.6,A -85,B 0,C 180,E1 -25202.199,E2 -25202.199} C_VEL
LIN {X 0,Y 275.119,Z 604.587,A -85,B 0,C 180,E1 -25205.112,E2 -25205.112} C_VEL
LIN {X 0,Y 276.507,Z 607.335,A -85,B 0,C 180,E1 -25207.276,E2 -25207.276} C_VEL
LIN {X 0,Y 278.849,Z 609.854,A -85,B 0,C 180,E1 -25210.127,E2 -25210.127} C_VEL
LIN {X 0,Y 281.89,Z 611.041,A -85,B 0,C 180,E1 -25212.922,E2 -25212.922} C_VEL
LIN {X 0,Y 283.774,Z 611.119,A -85,B 0,C 180,E1 -25214.29,E2 -25214.29} C_VEL
LIN {X 0,Y 288.178,Z 610.218,A -85,B 0,C 180,E1 -25216.958,E2 -25216.958} C_VEL
LIN {X 0,Y 292.994,Z 607.996,A -85,B 0,C 180,E1 -25219.553,E2 -25219.553} C_VEL
LIN {X 0,Y 298.297,Z 604.365,A -85,B 0,C 180,E1 -25222.068,E2 -25222.068} C_VEL
LIN {X 0,Y 304.268,Z 599.265,A -85,B 0,C 180,E1 -25224.479,E2 -25224.479} C_VEL
LIN {X 0,Y 309.016,Z 594.362,A -85,B 0,C 180,E1 -25226.232,E2 -25226.232} C_VEL
LIN {X 0,Y 314.869,Z 587.469,A -85,B 0,C 180,E1 -25228.211,E2 -25228.211} C_VEL
LIN {X 0,Y 321.213,Z 578.888,A -85,B 0,C 180,E1 -25230.102,E2 -25230.102} C_VEL
LIN {X 0,Y 327.913,Z 568.447,A -85,B 0,C 180,E1 -25231.916,E2 -25231.916} C_VEL
LIN {X 0,Y 333.868,Z 557.59,A -85,B 0,C 180,E1 -25233.416,E2 -25233.416} C_VEL
LIN {X 0,Y 339,Z 546.96,A -85,B 0,C 180,E1 -25234.625,E2 -25234.625} C_VEL
LIN {X 0,Y 344.1,Z 534.325,A -85,B 0,C 180,E1 -25235.819,E2 -25235.819} C_VEL
LIN {X 0,Y 348.824,Z 520.38,A -85,B 0,C 180,E1 -25236.862,E2 -25236.862} C_VEL
LIN {X 0,Y 352.585,Z 506.454,A -85,B 0,C 180,E1 -25237.698,E2 -25237.698} C_VEL
LIN {X 0,Y 357.63,Z 482.641,A -85,B 0,C 180,E1 -25238.728,E2 -25238.728} C_VEL
LIN {X 0,Y 361.328,Z 465.77,A -85,B 0,C 180,E1 -25239.354,E2 -25239.354} C_VEL
LIN {X 0,Y 360.678,Z 463.807,A -85,B 0,C 180,E1 -25240.659,E2 -25240.659} C_VEL
LIN {X 0,Y 360.001,Z 462.889,A -85,B 0,C 180,E1 -25242.92,E2 -25242.92} C_VEL
LIN {X 0,Y 360.159,Z 463.19,A -85,B 0,C 180,E1 -25244.93,E2 -25244.93} C_VEL
LIN {X 0,Y 360.592,Z 464.074,A -85,B 0,C 180,E1 -25246.199,E2 -25246.199} C_VEL
LIN {X 0,Y 360.291,Z 465.933,A -85,B 0,C 180,E1 -25246.439,E2 -25246.439} C_VEL
LIN {X 0,Y 357.177,Z 483.331,A -85,B 0,C 180,E1 -25247.947,E2 -25247.947} C_VEL
LIN {X 0,Y 354.741,Z 497.615,A -85,B 0,C 180,E1 -25248.994,E2 -25248.994} C_VEL
LIN {X 0,Y 353.366,Z 504.972,A -85,B 0,C 180,E1 -25249.395,E2 -25249.395} C_VEL
LIN {X 0,Y 348.716,Z 525.712,A -85,B 0,C 180,E1 -25250.142,E2 -25250.142} C_VEL
LIN {X 0,Y 343.899,Z 541.918,A -85,B 0,C 180,E1 -25250.846,E2 -25250.846} C_VEL
LIN {X 0,Y 337.15,Z 559.87,A -85,B 0,C 180,E1 -25251.824,E2 -25251.824} C_VEL
LIN {X 0,Y 330.638,Z 574.301,A -85,B 0,C 180,E1 -25252.86,E2 -25252.86} C_VEL
LIN {X 0,Y 323.278,Z 588.573,A -85,B 0,C 180,E1 -25254.196,E2 -25254.196} C_VEL
LIN {X 0,Y 316.36,Z 600.505,A -85,B 0,C 180,E1 -25255.626,E2 -25255.626} C_VEL
LIN {X 0,Y 308.845,Z 612.139,A -85,B 0,C 180,E1 -25257.409,E2 -25257.409} C_VEL
LIN {X 0,Y 302.934,Z 620.629,A -85,B 0,C 180,E1 -25259.038,E2 -25259.038} C_VEL
LIN {X 0,Y 295.84,Z 630.113,A -85,B 0,C 180,E1 -25261.35,E2 -25261.35} C_VEL
LIN {X 0,Y 290.359,Z 636.972,A -85,B 0,C 180,E1 -25263.494,E2 -25263.494} C_VEL
LIN {X 0,Y 284.991,Z 643.368,A -85,B 0,C 180,E1 -25266.075,E2 -25266.075} C_VEL
LIN {X 0,Y 280.434,Z 648.372,A -85,B 0,C 180,E1 -25268.766,E2 -25268.766} C_VEL
LIN {X 0,Y 277.694,Z 651.242,A -85,B 0,C 180,E1 -25270.858,E2 -25270.858} C_VEL
LIN {X 0,Y 275.118,Z 654.062,A -85,B 0,C 180,E1 -25273.736,E2 -25273.736} C_VEL
LIN {X 0,Y 273.387,Z 655.73,A -85,B 0,C 180,E1 -25276.804,E2 -25276.804} C_VEL
LIN {X 0,Y 273.124,Z 656.251,A -85,B 0,C 180,E1 -25277.667,E2 -25277.667} C_VEL
LIN {X 0,Y 272.859,Z 660.509,A -85,B 0,C 180,E1 -25280.767,E2 -25280.767} C_VEL
LIN {X 0,Y 272.883,Z 660.836,A -85,B 0,C 180,E1 -25281.047,E2 -25281.047} C_VEL
LIN {X 0,Y 272.505,Z 671.016,A -85,B 0,C 180,E1 -25283.358,E2 -25283.358} C_VEL
LIN {X 0,Y 272.403,Z 679.127,A -85,B 0,C 180,E1 -25285.576,E2 -25285.576} C_VEL
LIN {X 0,Y 272.202,Z 685.755,A -85,B 0,C 180,E1 -25287.788,E2 -25287.788} C_VEL
LIN {X 0,Y 272.112,Z 691.232,A -85,B 0,C 180,E1 -25290,E2 -25290} C_VEL
LIN {X 0,Y 271.839,Z 696.881,A -85,B 0,C 180,E1 -25292.954,E2 -25292.954} C_VEL
LIN {X 0,Y 271.913,Z 700.988,A -85,B 0,C 180,E1 -25295.914,E2 -25295.914} C_VEL
LIN {X 0,Y 272.519,Z 703.707,A -85,B 0,C 180,E1 -25298.871,E2 -25298.871} C_VEL
LIN {X 0,Y 274.075,Z 705.157,A -85,B 0,C 180,E1 -25301.797,E2 -25301.797} C_VEL
LIN {X 0,Y 276.404,Z 705.344,A -85,B 0,C 180,E1 -25304.679,E2 -25304.679} C_VEL
LIN {X 0,Y 279.726,Z 704.267,A -85,B 0,C 180,E1 -25307.487,E2 -25307.487} C_VEL
LIN {X 0,Y 283.495,Z 701.953,A -85,B 0,C 180,E1 -25310.237,E2 -25310.237} C_VEL
LIN {X 0,Y 288.29,Z 698.326,A -85,B 0,C 180,E1 -25312.876,E2 -25312.876} C_VEL
LIN {X 0,Y 293.919,Z 693.309,A -85,B 0,C 180,E1 -25315.402,E2 -25315.402} C_VEL
LIN {X 0,Y 300.212,Z 686.812,A -85,B 0,C 180,E1 -25317.816,E2 -25317.816} C_VEL
LIN {X 0,Y 306.321,Z 679.736,A -85,B 0,C 180,E1 -25319.824,E2 -25319.824} C_VEL
LIN {X 0,Y 313.782,Z 669.974,A -85,B 0,C 180,E1 -25321.977,E2 -25321.977} C_VEL
LIN {X 0,Y 321.069,Z 659.319,A -85,B 0,C 180,E1 -25323.801,E2 -25323.801} C_VEL
LIN {X 0,Y 328.166,Z 647.559,A -85,B 0,C 180,E1 -25325.377,E2 -25325.377} C_VEL
LIN {X 0,Y 334.536,Z 635.621,A -85,B 0,C 180,E1 -25326.636,E2 -25326.636} C_VEL
LIN {X 0,Y 339.986,Z 624.117,A -85,B 0,C 180,E1 -25327.614,E2 -25327.614} C_VEL
LIN {X 0,Y 345.704,Z 610.229,A -85,B 0,C 180,E1 -25328.538,E2 -25328.538} C_VEL
LIN {X 0,Y 350.682,Z 595.758,A -85,B 0,C 180,E1 -25329.266,E2 -25329.266} C_VEL
LIN {X 0,Y 355.294,Z 578.812,A -85,B 0,C 180,E1 -25329.938,E2 -25329.938} C_VEL
LIN {X 0,Y 371.871,Z 507.617,A -85,B 0,C 180,E1 -25332.419,E2 -25332.419} C_VEL
LIN {X 0,Y 373.1,Z 501.951,A -85,B 0,C 180,E1 -25332.811,E2 -25332.811} C_VEL
LIN {X 0,Y 372.411,Z 502.417,A -85,B 0,C 180,E1 -25334.532,E2 -25334.532} C_VEL
LIN {X 0,Y 372.018,Z 504.844,A -85,B 0,C 180,E1 -25336.366,E2 -25336.366} C_VEL
LIN {X 0,Y 371.91,Z 505.755,A -85,B 0,C 180,E1 -25336.68,E2 -25336.68} C_VEL
LIN {X 0,Y 369.797,Z 516.339,A -85,B 0,C 180,E1 -25337.803,E2 -25337.803} C_VEL
LIN {X 0,Y 369.305,Z 518.612,A -85,B 0,C 180,E1 -25337.952,E2 -25337.952} C_VEL
LIN {X 0,Y 353.581,Z 586.024,A -85,B 0,C 180,E1 -25340.292,E2 -25340.292} C_VEL
LIN {X 0,Y 348.912,Z 601.353,A -85,B 0,C 180,E1 -25340.961,E2 -25340.961} C_VEL
LIN {X 0,Y 343.153,Z 616.727,A -85,B 0,C 180,E1 -25341.869,E2 -25341.869} C_VEL
LIN {X 0,Y 337.629,Z 629.28,A -85,B 0,C 180,E1 -25342.827,E2 -25342.827} C_VEL
LIN {X 0,Y 330.624,Z 643.112,A -85,B 0,C 180,E1 -25344.18,E2 -25344.18} C_VEL
LIN {X 0,Y 324.239,Z 654.13,A -85,B 0,C 180,E1 -25345.554,E2 -25345.554} C_VEL
LIN {X 0,Y 318.177,Z 663.501,A -85,B 0,C 180,E1 -25346.986,E2 -25346.986} C_VEL
LIN {X 0,Y 311.233,Z 673.151,A -85,B 0,C 180,E1 -25348.827,E2 -25348.827} C_VEL
LIN {X 0,Y 304.804,Z 681.185,A -85,B 0,C 180,E1 -25350.77,E2 -25350.77} C_VEL
LIN {X 0,Y 298.859,Z 687.834,A -85,B 0,C 180,E1 -25352.805,E2 -25352.805} C_VEL
LIN {X 0,Y 292.797,Z 693.908,A -85,B 0,C 180,E1 -25355.251,E2 -25355.251} C_VEL
LIN {X 0,Y 288.723,Z 697.506,A -85,B 0,C 180,E1 -25357.16,E2 -25357.16} C_VEL
LIN {X 0,Y 283.824,Z 701.118,A -85,B 0,C 180,E1 -25359.788,E2 -25359.788} C_VEL
LIN {X 0,Y 279.977,Z 703.406,A -85,B 0,C 180,E1 -25362.53,E2 -25362.53} C_VEL
LIN {X 0,Y 276.622,Z 704.458,A -85,B 0,C 180,E1 -25365.333,E2 -25365.333} C_VEL
LIN {X 0,Y 274.219,Z 704.249,A -85,B 0,C 180,E1 -25368.209,E2 -25368.209} C_VEL
LIN {X 0,Y 272.598,Z 702.782,A -85,B 0,C 180,E1 -25371.132,E2 -25371.132} C_VEL
LIN {X 0,Y 271.923,Z 700.048,A -85,B 0,C 180,E1 -25374.086,E2 -25374.086} C_VEL
LIN {X 0,Y 271.693,Z 695.929,A -85,B 0,C 180,E1 -25377.045,E2 -25377.045} C_VEL
LIN {X 0,Y 271.879,Z 691.9,A -85,B 0,C 180,E1 -25379.262,E2 -25379.262} C_VEL
LIN {X 0,Y 272.011,Z 686.811,A -85,B 0,C 180,E1 -25381.476,E2 -25381.476} C_VEL
LIN {X 0,Y 272.301,Z 679.532,A -85,B 0,C 180,E1 -25384.057,E2 -25384.057} C_VEL
LIN {X 0,Y 272.496,Z 670.338,A -85,B 0,C 180,E1 -25386.643,E2 -25386.643} C_VEL
LIN {X 0,Y 272.948,Z 660.784,A -85,B 0,C 180,E1 -25388.858,E2 -25388.858} C_VEL
LIN {X 0,Y 273.506,Z 649.232,A -85,B 0,C 180,E1 -25391.074,E2 -25391.074} C_VEL
LIN {X 0,Y 274.227,Z 637.608,A -85,B 0,C 180,E1 -25392.915,E2 -25392.915} C_VEL
LIN {X 0,Y 275.1,Z 623.331,A -85,B 0,C 180,E1 -25394.751,E2 -25394.751} C_VEL
LIN {X 0,Y 275.969,Z 609.219,A -85,B 0,C 180,E1 -25396.213,E2 -25396.213} C_VEL
LIN {X 0,Y 276.686,Z 594.464,A -85,B 0,C 180,E1 -25397.4,E2 -25397.4} C_VEL
LIN {X 0,Y 277.423,Z 578.672,A -85,B 0,C 180,E1 -25398.35,E2 -25398.35} C_VEL
LIN {X 0,Y 281.067,Z 478.635,A -85,B 0,C 180,E1 -25402.769,E2 -25402.769} C_VEL
LIN {X 0,Y 278.98,Z 450.492,A -85,B 0,C 180,E1 -25404.03,E2 -25404.03} C_VEL
LIN {X 0,Y 278.78,Z 439.514,A -85,B 0,C 180,E1 -25404.542,E2 -25404.542} C_VEL
LIN {X 0,Y 281.627,Z 412.456,A -85,B 0,C 180,E1 -25409.211,E2 -25409.211} C_VEL
LIN {X 0,Y 282.762,Z 402.439,A -85,B 0,C 180,E1 -25410.932,E2 -25410.932} C_VEL
LIN {X 0,Y 279.433,Z 386.674,A -85,B 0,C 180,E1 -25413.88,E2 -25413.88} C_VEL
LIN {X 0,Y 275.445,Z 368.551,A -85,B 0,C 180,E1 -25417.377,E2 -25417.377} C_VEL
LIN {X 0,Y 274.399,Z 363.863,A -85,B 0,C 180,E1 -25418.331,E2 -25418.331} C_VEL
LIN {X 0,Y 274.329,Z 363.868,A -85,B 0,C 180,E1 -25422.23,E2 -25422.23} C_VEL
LIN {X 0,Y 274.373,Z 363.857,A -85,B 0,C 180,E1 -25425.628,E2 -25425.628} C_VEL
LIN {X 0,Y 274.335,Z 363.861,A -85,B 0,C 180,E1 -25429.995,E2 -25429.995} C_VEL
LIN {X 0,Y 274.347,Z 363.861,A -85,B 0,C 180,E1 -25434.04,E2 -25434.04} C_VEL
LIN {X 0,Y 274.347,Z 363.848,A -85,B 0,C 180,E1 -25437.578,E2 -25437.578} C_VEL
LIN {X 0,Y 274.394,Z 363.86,A -85,B 0,C 180,E1 -25441.855,E2 -25441.855} C_VEL
LIN {X 0,Y 275.42,Z 366.768,A -85,B 0,C 180,E1 -25442.103,E2 -25442.103} C_VEL
LIN {X 0,Y 281.751,Z 378.157,A -85,B 0,C 180,E1 -25443.217,E2 -25443.217} C_VEL
LIN {X 0,Y 290.189,Z 395.508,A -85,B 0,C 180,E1 -25444.67,E2 -25444.67} C_VEL
LIN {X 0,Y 294.537,Z 405.563,A -85,B 0,C 180,E1 -25445.409,E2 -25445.409} C_VEL
LIN {X 0,Y 292.743,Z 467.339,A -85,B 0,C 180,E1 -25446.896,E2 -25446.896} C_VEL
LIN {X 0,Y 292.336,Z 484.943,A -85,B 0,C 180,E1 -25447.425,E2 -25447.425} C_VEL
LIN {X 0,Y 291.598,Z 499.381,A -85,B 0,C 180,E1 -25448.141,E2 -25448.141} C_VEL
LIN {X 0,Y 290.35,Z 512.77,A -85,B 0,C 180,E1 -25449.063,E2 -25449.063} C_VEL
LIN {X 0,Y 288.872,Z 524.875,A -85,B 0,C 180,E1 -25450.156,E2 -25450.156} C_VEL
LIN {X 0,Y 287.328,Z 536.771,A -85,B 0,C 180,E1 -25451.524,E2 -25451.524} C_VEL
LIN {X 0,Y 285.463,Z 547.856,A -85,B 0,C 180,E1 -25453.078,E2 -25453.078} C_VEL
LIN {X 0,Y 283.226,Z 559.071,A -85,B 0,C 180,E1 -25455.005,E2 -25455.005} C_VEL
LIN {X 0,Y 281.099,Z 568.715,A -85,B 0,C 180,E1 -25457.041,E2 -25457.041} C_VEL
LIN {X 0,Y 279.258,Z 576.941,A -85,B 0,C 180,E1 -25459.157,E2 -25459.157} C_VEL
LIN {X 0,Y 277.728,Z 583.804,A -85,B 0,C 180,E1 -25461.297,E2 -25461.297} C_VEL
LIN {X 0,Y 276.329,Z 589.493,A -85,B 0,C 180,E1 -25463.45,E2 -25463.45} C_VEL
LIN {X 0,Y 275.042,Z 595.561,A -85,B 0,C 180,E1 -25466.35,E2 -25466.35} C_VEL
LIN {X 0,Y 274.383,Z 599.02,A -85,B 0,C 180,E1 -25468.537,E2 -25468.537} C_VEL
LIN {X 0,Y 273.752,Z 602.438,A -85,B 0,C 180,E1 -25471.466,E2 -25471.466} C_VEL
LIN {X 0,Y 273.753,Z 604.484,A -85,B 0,C 180,E1 -25474.403,E2 -25474.403} C_VEL
LIN {X 0,Y 273.966,Z 605.254,A -85,B 0,C 180,E1 -25477.345,E2 -25477.345} C_VEL
LIN {X 0,Y 274.623,Z 604.728,A -85,B 0,C 180,E1 -25480.285,E2 -25480.285} C_VEL
LIN {X 0,Y 275.66,Z 602.89,A -85,B 0,C 180,E1 -25483.22,E2 -25483.22} C_VEL
LIN {X 0,Y 277.41,Z 599.651,A -85,B 0,C 180,E1 -25486.126,E2 -25486.126} C_VEL
LIN {X 0,Y 279.534,Z 594.946,A -85,B 0,C 180,E1 -25489.011,E2 -25489.011} C_VEL
LIN {X 0,Y 282.205,Z 588.61,A -85,B 0,C 180,E1 -25491.858,E2 -25491.858} C_VEL
LIN {X 0,Y 285.097,Z 581.097,A -85,B 0,C 180,E1 -25494.451,E2 -25494.451} C_VEL
LIN {X 0,Y 288.035,Z 572.717,A -85,B 0,C 180,E1 -25496.737,E2 -25496.737} C_VEL
LIN {X 0,Y 291.054,Z 563.419,A -85,B 0,C 180,E1 -25498.772,E2 -25498.772} C_VEL
LIN {X 0,Y 294.099,Z 552.354,A -85,B 0,C 180,E1 -25500.741,E2 -25500.741} C_VEL
LIN {X 0,Y 296.749,Z 541.649,A -85,B 0,C 180,E1 -25502.279,E2 -25502.279} C_VEL
LIN {X 0,Y 299.516,Z 528.9,A -85,B 0,C 180,E1 -25503.74,E2 -25503.74} C_VEL
LIN {X 0,Y 301.455,Z 516.39,A -85,B 0,C 180,E1 -25504.902,E2 -25504.902} C_VEL
LIN {X 0,Y 303.151,Z 502.434,A -85,B 0,C 180,E1 -25505.891,E2 -25505.891} C_VEL
LIN {X 0,Y 304.328,Z 488.086,A -85,B 0,C 180,E1 -25506.614,E2 -25506.614} C_VEL
LIN {X 0,Y 304.87,Z 472.949,A -85,B 0,C 180,E1 -25507.104,E2 -25507.104} C_VEL
LIN {X 0,Y 306.965,Z 420.262,A -85,B 0,C 180,E1 -25508.315,E2 -25508.315} C_VEL
LIN {X 0,Y 297.986,Z 402.616,A -85,B 0,C 180,E1 -25510.121,E2 -25510.121} C_VEL
LIN {X 0,Y 289.327,Z 387.675,A -85,B 0,C 180,E1 -25511.951,E2 -25511.951} C_VEL
LIN {X 0,Y 281.835,Z 376.009,A -85,B 0,C 180,E1 -25513.627,E2 -25513.627} C_VEL
LIN {X 0,Y 279.121,Z 372.093,A -85,B 0,C 180,E1 -25514.258,E2 -25514.258} C_VEL
LIN {X 0,Y 276.658,Z 368.345,A -85,B 0,C 180,E1 -25514.853,E2 -25514.853} C_VEL
LIN {X 0,Y 274.903,Z 365.978,A -85,B 0,C 180,E1 -25515.277,E2 -25515.277} C_VEL
LIN {X 0,Y 274.299,Z 363.872,A -85,B 0,C 180,E1 -25515.502,E2 -25515.502} C_VEL
LIN {X 0,Y 274.302,Z 363.872,A -85,B 0,C 180,E1 -25520.002,E2 -25520.002} C_VEL
LIN {X 0,Y 274.338,Z 363.818,A -85,B 0,C 180,E1 -25524.038,E2 -25524.038} C_VEL
LIN {X 0,Y 274.334,Z 363.868,A -85,B 0,C 180,E1 -25527.575,E2 -25527.575} C_VEL
LIN {X 0,Y 274.332,Z 363.866,A -85,B 0,C 180,E1 -25530.979,E2 -25530.979} C_VEL
LIN {X 0,Y 274.37,Z 363.849,A -85,B 0,C 180,E1 -25534.278,E2 -25534.278} C_VEL
LIN {X 0,Y 274.475,Z 363.852,A -85,B 0,C 180,E1 -25536.096,E2 -25536.096} C_VEL
LIN {X 0,Y 279.736,Z 386.043,A -85,B 0,C 180,E1 -25537.155,E2 -25537.155} C_VEL
LIN {X 0,Y 280.258,Z 388.844,A -85,B 0,C 180,E1 -25537.284,E2 -25537.284} C_VEL
